(* IEC 61131-3 sources: AXOpen/src/showcase/app/src/IO (part 3) *)

	TYPE
        {S7.extern=ReadWrite}
        {#ix-attr:[Container(Layout.Wrap)]}
	    cognex_insight_7600_ResultData_128_Input_Layout : STRUCT
	        Signals_0 AT %B0 : WORD;
	        Signals_1 AT %B2 : WORD;
	        Signals_2 AT %B4 : ARRAY[0..127] OF BYTE;
	    END_STRUCT;
	END_TYPE

	TYPE
        {S7.extern=ReadWrite}
        {#ix-attr:[Container(Layout.Wrap)]}
	    cognex_insight_7600_SoftEvent_Control_Input_Layout : STRUCT
	        Signals_0 AT %X0.0 : BOOL;
	        Signals_1 AT %X0.1 : BOOL;
	        Signals_2 AT %X0.2 : BOOL;
	        Signals_3 AT %X0.3 : BOOL;
	        Signals_4 AT %X0.4 : BOOL;
	        Signals_5 AT %X0.5 : BOOL;
	        Signals_6 AT %X0.6 : BOOL;
	        Signals_7 AT %X0.7 : BOOL;
	    END_STRUCT;
	END_TYPE

	TYPE
        {S7.extern=ReadWrite}
        {#ix-attr:[Container(Layout.Wrap)]}
	    cognex_insight_7600_SoftEvent_Control_Output_Layout : STRUCT
	        Signals_8 AT %X0.0 : BOOL;
	        Signals_9 AT %X0.1 : BOOL;
	        Signals_10 AT %X0.2 : BOOL;
	        Signals_11 AT %X0.3 : BOOL;
	        Signals_12 AT %X0.4 : BOOL;
	        Signals_13 AT %X0.5 : BOOL;
	        Signals_14 AT %X0.6 : BOOL;
	        Signals_15 AT %X0.7 : BOOL;
	    END_STRUCT;
	END_TYPE

	TYPE
        {S7.extern=ReadWrite}
        {#ix-attr:[Container(Layout.Wrap)]}
	    cognex_insight_7600_UserData_128_Output_Layout : STRUCT
	        Signals_0 AT %B0 : ARRAY[0..127] OF BYTE;
	    END_STRUCT;
	END_TYPE

	TYPE
        {S7.extern=ReadWrite}
        {#ix-attr:[Container(Layout.Wrap)]}
	    desoutter_cvic_ii_Input_1_byte_1_Input_Layout : STRUCT
	        Signals_0 AT %B0 : BYTE;
	    END_STRUCT;
	END_TYPE

	TYPE
        {S7.extern=ReadWrite}
        {#ix-attr:[Container(Layout.Wrap)]}
	    desoutter_cvic_ii_Input_1_byte_2_Input_Layout : STRUCT
	        Signals_0 AT %B0 : BYTE;
	    END_STRUCT;
	END_TYPE

	TYPE
        {S7.extern=ReadWrite}
        {#ix-attr:[Container(Layout.Wrap)]}
	    desoutter_cvic_ii_Input_1_word_1_Input_Layout : STRUCT
	        Signals_0 AT %B0 : WORD;
	    END_STRUCT;
	END_TYPE

	TYPE
        {S7.extern=ReadWrite}
        {#ix-attr:[Container(Layout.Wrap)]}
	    desoutter_cvic_ii_Input_1_word_2_Input_Layout : STRUCT
	        Signals_0 AT %B0 : WORD;
	    END_STRUCT;
	END_TYPE

	TYPE
        {S7.extern=ReadWrite}
        {#ix-attr:[Container(Layout.Wrap)]}
	    desoutter_cvic_ii_Input_2_word_1_Input_Layout : STRUCT
	        Signals_0 AT %B0 : DWORD;
	    END_STRUCT;
	END_TYPE

	TYPE
        {S7.extern=ReadWrite}
        {#ix-attr:[Container(Layout.Wrap)]}
	    desoutter_cvic_ii_Input_2_word_2_Input_Layout : STRUCT
	        Signals_0 AT %B0 : DWORD;
	    END_STRUCT;
	END_TYPE

	TYPE
        {S7.extern=ReadWrite}
        {#ix-attr:[Container(Layout.Wrap)]}
	    desoutter_cvic_ii_Output_1_byte_1_Output_Layout : STRUCT
	        Signals_0 AT %B0 : BYTE;
	    END_STRUCT;
	END_TYPE

	TYPE
        {S7.extern=ReadWrite}
        {#ix-attr:[Container(Layout.Wrap)]}
	    desoutter_cvic_ii_Output_1_byte_2_Output_Layout : STRUCT
	        Signals_0 AT %B0 : BYTE;
	    END_STRUCT;
	END_TYPE

	TYPE
        {S7.extern=ReadWrite}
        {#ix-attr:[Container(Layout.Wrap)]}
	    dukaneiqauto_iQ_to_PLC_Inputs_Input_Layout : STRUCT
	        Signals_0 AT %B0 : DWORD;
	        Signals_1 AT %B4 : DWORD;
	        Signals_2 AT %B8 : DWORD;
	        Signals_3 AT %B12 : DWORD;
	        Signals_4 AT %B16 : DWORD;
	        Signals_5 AT %B20 : DWORD;
	        Signals_6 AT %B24 : DWORD;
	        Signals_7 AT %B28 : DWORD;
	        Signals_8 AT %B32 : DWORD;
	        Signals_9 AT %B36 : DWORD;
	        Signals_10 AT %B40 : DWORD;
	        Signals_11 AT %B44 : DWORD;
	        Signals_12 AT %B48 : DWORD;
	        Signals_13 AT %B52 : DWORD;
	        Signals_14 AT %B56 : DWORD;
	        Signals_15 AT %B60 : DWORD;
	        Signals_16 AT %B64 : DWORD;
	        Signals_17 AT %B68 : DWORD;
	        Signals_18 AT %B72 : DWORD;
	        Signals_19 AT %B76 : DWORD;
	        Signals_20 AT %B80 : DWORD;
	        Signals_21 AT %B84 : DWORD;
	        Signals_22 AT %B88 : DWORD;
	        Signals_23 AT %B92 : DWORD;
	        Signals_24 AT %B96 : DWORD;
	        Signals_25 AT %B100 : DWORD;
	        Signals_26 AT %B104 : DWORD;
	        Signals_27 AT %B108 : DWORD;
	        Signals_28 AT %B112 : DWORD;
	        Signals_29 AT %B116 : DWORD;
	        Signals_30 AT %B120 : DWORD;
	        Signals_31 AT %B124 : DWORD;
	        Signals_32 AT %B128 : DWORD;
	        Signals_33 AT %B132 : DWORD;
	        Signals_34 AT %B136 : DWORD;
	    END_STRUCT;
	END_TYPE

	TYPE
        {S7.extern=ReadWrite}
        {#ix-attr:[Container(Layout.Wrap)]}
	    dukaneiqauto_PLC_to_iQ_Outputs_Output_Layout : STRUCT
	        Signals_0 AT %B0 : DWORD;
	        Signals_1 AT %B4 : DWORD;
	        Signals_2 AT %B8 : DWORD;
	        Signals_3 AT %B12 : DWORD;
	        Signals_4 AT %B16 : DWORD;
	    END_STRUCT;
	END_TYPE

	TYPE
        {S7.extern=ReadWrite}
        {#ix-attr:[Container(Layout.Wrap)]}
	    et200sp_CM_4xIO_Link_RF200_CM_4xIO_Link_V2_2_144I_128O_1_Input_Layout : STRUCT
	        Signals_0 AT %B0 : BYTE;
	        Signals_1 AT %B1 : BYTE;
	        Signals_2 AT %B2 : BYTE;
	        Signals_3 AT %B3 : BYTE;
	        Signals_4 AT %B4 : BYTE;
	        Signals_5 AT %B5 : BYTE;
	        Signals_6 AT %B6 : BYTE;
	        Signals_7 AT %B7 : BYTE;
	        Signals_8 AT %B8 : BYTE;
	        Signals_9 AT %B9 : BYTE;
	        Signals_10 AT %B10 : BYTE;
	        Signals_11 AT %B11 : BYTE;
	        Signals_12 AT %B12 : BYTE;
	        Signals_13 AT %B13 : BYTE;
	        Signals_14 AT %B14 : BYTE;
	        Signals_15 AT %B15 : BYTE;
	        Signals_16 AT %B16 : BYTE;
	        Signals_17 AT %B17 : BYTE;
	        Signals_18 AT %B18 : BYTE;
	        Signals_19 AT %B19 : BYTE;
	        Signals_20 AT %B20 : BYTE;
	        Signals_21 AT %B21 : BYTE;
	        Signals_22 AT %B22 : BYTE;
	        Signals_23 AT %B23 : BYTE;
	        Signals_24 AT %B24 : BYTE;
	        Signals_25 AT %B25 : BYTE;
	        Signals_26 AT %B26 : BYTE;
	        Signals_27 AT %B27 : BYTE;
	        Signals_28 AT %B28 : BYTE;
	        Signals_29 AT %B29 : BYTE;
	        Signals_30 AT %B30 : BYTE;
	        Signals_31 AT %B31 : BYTE;
	        Signals_32 AT %B32 : BYTE;
	        Signals_33 AT %B33 : BYTE;
	        Signals_34 AT %B34 : BYTE;
	        Signals_35 AT %B35 : BYTE;
	        Signals_36 AT %B36 : BYTE;
	        Signals_37 AT %B37 : BYTE;
	        Signals_38 AT %B38 : BYTE;
	        Signals_39 AT %B39 : BYTE;
	        Signals_40 AT %B40 : BYTE;
	        Signals_41 AT %B41 : BYTE;
	        Signals_42 AT %B42 : BYTE;
	        Signals_43 AT %B43 : BYTE;
	        Signals_44 AT %B44 : BYTE;
	        Signals_45 AT %B45 : BYTE;
	        Signals_46 AT %B46 : BYTE;
	        Signals_47 AT %B47 : BYTE;
	        Signals_48 AT %B48 : BYTE;
	        Signals_49 AT %B49 : BYTE;
	        Signals_50 AT %B50 : BYTE;
	        Signals_51 AT %B51 : BYTE;
	        Signals_52 AT %B52 : BYTE;
	        Signals_53 AT %B53 : BYTE;
	        Signals_54 AT %B54 : BYTE;
	        Signals_55 AT %B55 : BYTE;
	        Signals_56 AT %B56 : BYTE;
	        Signals_57 AT %B57 : BYTE;
	        Signals_58 AT %B58 : BYTE;
	        Signals_59 AT %B59 : BYTE;
	        Signals_60 AT %B60 : BYTE;
	        Signals_61 AT %B61 : BYTE;
	        Signals_62 AT %B62 : BYTE;
	        Signals_63 AT %B63 : BYTE;
	        Signals_64 AT %B64 : BYTE;
	        Signals_65 AT %B65 : BYTE;
	        Signals_66 AT %B66 : BYTE;
	        Signals_67 AT %B67 : BYTE;
	        Signals_68 AT %B68 : BYTE;
	        Signals_69 AT %B69 : BYTE;
	        Signals_70 AT %B70 : BYTE;
	        Signals_71 AT %B71 : BYTE;
	        Signals_72 AT %B72 : BYTE;
	        Signals_73 AT %B73 : BYTE;
	        Signals_74 AT %B74 : BYTE;
	        Signals_75 AT %B75 : BYTE;
	        Signals_76 AT %B76 : BYTE;
	        Signals_77 AT %B77 : BYTE;
	        Signals_78 AT %B78 : BYTE;
	        Signals_79 AT %B79 : BYTE;
	        Signals_80 AT %B80 : BYTE;
	        Signals_81 AT %B81 : BYTE;
	        Signals_82 AT %B82 : BYTE;
	        Signals_83 AT %B83 : BYTE;
	        Signals_84 AT %B84 : BYTE;
	        Signals_85 AT %B85 : BYTE;
	        Signals_86 AT %B86 : BYTE;
	        Signals_87 AT %B87 : BYTE;
	        Signals_88 AT %B88 : BYTE;
	        Signals_89 AT %B89 : BYTE;
	        Signals_90 AT %B90 : BYTE;
	        Signals_91 AT %B91 : BYTE;
	        Signals_92 AT %B92 : BYTE;
	        Signals_93 AT %B93 : BYTE;
	        Signals_94 AT %B94 : BYTE;
	        Signals_95 AT %B95 : BYTE;
	        Signals_96 AT %B96 : BYTE;
	        Signals_97 AT %B97 : BYTE;
	        Signals_98 AT %B98 : BYTE;
	        Signals_99 AT %B99 : BYTE;
	        Signals_100 AT %B100 : BYTE;
	        Signals_101 AT %B101 : BYTE;
	        Signals_102 AT %B102 : BYTE;
	        Signals_103 AT %B103 : BYTE;
	        Signals_104 AT %B104 : BYTE;
	        Signals_105 AT %B105 : BYTE;
	        Signals_106 AT %B106 : BYTE;
	        Signals_107 AT %B107 : BYTE;
	        Signals_108 AT %B108 : BYTE;
	        Signals_109 AT %B109 : BYTE;
	        Signals_110 AT %B110 : BYTE;
	        Signals_111 AT %B111 : BYTE;
	        Signals_112 AT %B112 : BYTE;
	        Signals_113 AT %B113 : BYTE;
	        Signals_114 AT %B114 : BYTE;
	        Signals_115 AT %B115 : BYTE;
	        Signals_116 AT %B116 : BYTE;
	        Signals_117 AT %B117 : BYTE;
	        Signals_118 AT %B118 : BYTE;
	        Signals_119 AT %B119 : BYTE;
	        Signals_120 AT %B120 : BYTE;
	        Signals_121 AT %B121 : BYTE;
	        Signals_122 AT %B122 : BYTE;
	        Signals_123 AT %B123 : BYTE;
	        Signals_124 AT %B124 : BYTE;
	        Signals_125 AT %B125 : BYTE;
	        Signals_126 AT %B126 : BYTE;
	        Signals_127 AT %B127 : BYTE;
	        Signals_128 AT %B128 : BYTE;
	        Signals_129 AT %B129 : BYTE;
	        Signals_130 AT %B130 : BYTE;
	        Signals_131 AT %B131 : BYTE;
	        Signals_132 AT %B132 : BYTE;
	        Signals_133 AT %B133 : BYTE;
	        Signals_134 AT %B134 : BYTE;
	        Signals_135 AT %B135 : BYTE;
	        Signals_136 AT %B136 : BYTE;
	        Signals_137 AT %B137 : BYTE;
	        Signals_138 AT %B138 : BYTE;
	        Signals_139 AT %B139 : BYTE;
	        Signals_140 AT %B140 : BYTE;
	        Signals_141 AT %B141 : BYTE;
	        Signals_142 AT %B142 : BYTE;
	        Signals_143 AT %B143 : BYTE;
	    END_STRUCT;
	END_TYPE

	TYPE
        {S7.extern=ReadWrite}
        {#ix-attr:[Container(Layout.Wrap)]}
	    et200sp_CM_4xIO_Link_RF200_CM_4xIO_Link_V2_2_144I_128O_1_Output_Layout : STRUCT
	        Signals_144 AT %B0 : BYTE;
	        Signals_145 AT %B1 : BYTE;
	        Signals_146 AT %B2 : BYTE;
	        Signals_147 AT %B3 : BYTE;
	        Signals_148 AT %B4 : BYTE;
	        Signals_149 AT %B5 : BYTE;
	        Signals_150 AT %B6 : BYTE;
	        Signals_151 AT %B7 : BYTE;
	        Signals_152 AT %B8 : BYTE;
	        Signals_153 AT %B9 : BYTE;
	        Signals_154 AT %B10 : BYTE;
	        Signals_155 AT %B11 : BYTE;
	        Signals_156 AT %B12 : BYTE;
	        Signals_157 AT %B13 : BYTE;
	        Signals_158 AT %B14 : BYTE;
	        Signals_159 AT %B15 : BYTE;
	        Signals_160 AT %B16 : BYTE;
	        Signals_161 AT %B17 : BYTE;
	        Signals_162 AT %B18 : BYTE;
	        Signals_163 AT %B19 : BYTE;
	        Signals_164 AT %B20 : BYTE;
	        Signals_165 AT %B21 : BYTE;
	        Signals_166 AT %B22 : BYTE;
	        Signals_167 AT %B23 : BYTE;
	        Signals_168 AT %B24 : BYTE;
	        Signals_169 AT %B25 : BYTE;
	        Signals_170 AT %B26 : BYTE;
	        Signals_171 AT %B27 : BYTE;
	        Signals_172 AT %B28 : BYTE;
	        Signals_173 AT %B29 : BYTE;
	        Signals_174 AT %B30 : BYTE;
	        Signals_175 AT %B31 : BYTE;
	        Signals_176 AT %B32 : BYTE;
	        Signals_177 AT %B33 : BYTE;
	        Signals_178 AT %B34 : BYTE;
	        Signals_179 AT %B35 : BYTE;
	        Signals_180 AT %B36 : BYTE;
	        Signals_181 AT %B37 : BYTE;
	        Signals_182 AT %B38 : BYTE;
	        Signals_183 AT %B39 : BYTE;
	        Signals_184 AT %B40 : BYTE;
	        Signals_185 AT %B41 : BYTE;
	        Signals_186 AT %B42 : BYTE;
	        Signals_187 AT %B43 : BYTE;
	        Signals_188 AT %B44 : BYTE;
	        Signals_189 AT %B45 : BYTE;
	        Signals_190 AT %B46 : BYTE;
	        Signals_191 AT %B47 : BYTE;
	        Signals_192 AT %B48 : BYTE;
	        Signals_193 AT %B49 : BYTE;
	        Signals_194 AT %B50 : BYTE;
	        Signals_195 AT %B51 : BYTE;
	        Signals_196 AT %B52 : BYTE;
	        Signals_197 AT %B53 : BYTE;
	        Signals_198 AT %B54 : BYTE;
	        Signals_199 AT %B55 : BYTE;
	        Signals_200 AT %B56 : BYTE;
	        Signals_201 AT %B57 : BYTE;
	        Signals_202 AT %B58 : BYTE;
	        Signals_203 AT %B59 : BYTE;
	        Signals_204 AT %B60 : BYTE;
	        Signals_205 AT %B61 : BYTE;
	        Signals_206 AT %B62 : BYTE;
	        Signals_207 AT %B63 : BYTE;
	        Signals_208 AT %B64 : BYTE;
	        Signals_209 AT %B65 : BYTE;
	        Signals_210 AT %B66 : BYTE;
	        Signals_211 AT %B67 : BYTE;
	        Signals_212 AT %B68 : BYTE;
	        Signals_213 AT %B69 : BYTE;
	        Signals_214 AT %B70 : BYTE;
	        Signals_215 AT %B71 : BYTE;
	        Signals_216 AT %B72 : BYTE;
	        Signals_217 AT %B73 : BYTE;
	        Signals_218 AT %B74 : BYTE;
	        Signals_219 AT %B75 : BYTE;
	        Signals_220 AT %B76 : BYTE;
	        Signals_221 AT %B77 : BYTE;
	        Signals_222 AT %B78 : BYTE;
	        Signals_223 AT %B79 : BYTE;
	        Signals_224 AT %B80 : BYTE;
	        Signals_225 AT %B81 : BYTE;
	        Signals_226 AT %B82 : BYTE;
	        Signals_227 AT %B83 : BYTE;
	        Signals_228 AT %B84 : BYTE;
	        Signals_229 AT %B85 : BYTE;
	        Signals_230 AT %B86 : BYTE;
	        Signals_231 AT %B87 : BYTE;
	        Signals_232 AT %B88 : BYTE;
	        Signals_233 AT %B89 : BYTE;
	        Signals_234 AT %B90 : BYTE;
	        Signals_235 AT %B91 : BYTE;
	        Signals_236 AT %B92 : BYTE;
	        Signals_237 AT %B93 : BYTE;
	        Signals_238 AT %B94 : BYTE;
	        Signals_239 AT %B95 : BYTE;
	        Signals_240 AT %B96 : BYTE;
	        Signals_241 AT %B97 : BYTE;
	        Signals_242 AT %B98 : BYTE;
	        Signals_243 AT %B99 : BYTE;
	        Signals_244 AT %B100 : BYTE;
	        Signals_245 AT %B101 : BYTE;
	        Signals_246 AT %B102 : BYTE;
	        Signals_247 AT %B103 : BYTE;
	        Signals_248 AT %B104 : BYTE;
	        Signals_249 AT %B105 : BYTE;
	        Signals_250 AT %B106 : BYTE;
	        Signals_251 AT %B107 : BYTE;
	        Signals_252 AT %B108 : BYTE;
	        Signals_253 AT %B109 : BYTE;
	        Signals_254 AT %B110 : BYTE;
	        Signals_255 AT %B111 : BYTE;
	        Signals_256 AT %B112 : BYTE;
	        Signals_257 AT %B113 : BYTE;
	        Signals_258 AT %B114 : BYTE;
	        Signals_259 AT %B115 : BYTE;
	        Signals_260 AT %B116 : BYTE;
	        Signals_261 AT %B117 : BYTE;
	        Signals_262 AT %B118 : BYTE;
	        Signals_263 AT %B119 : BYTE;
	        Signals_264 AT %B120 : BYTE;
	        Signals_265 AT %B121 : BYTE;
	        Signals_266 AT %B122 : BYTE;
	        Signals_267 AT %B123 : BYTE;
	        Signals_268 AT %B124 : BYTE;
	        Signals_269 AT %B125 : BYTE;
	        Signals_270 AT %B126 : BYTE;
	        Signals_271 AT %B127 : BYTE;
	    END_STRUCT;
	END_TYPE

	TYPE
        {S7.extern=ReadWrite}
        {#ix-attr:[Container(Layout.Wrap)]}
	    et200sp_CpPtp_Input_Layout : STRUCT
	        Signals_0 AT %B0 : BYTE;
	        Signals_1 AT %B1 : BYTE;
	        Signals_2 AT %B2 : BYTE;
	        Signals_3 AT %B3 : BYTE;
	        Signals_4 AT %B4 : BYTE;
	        Signals_5 AT %B5 : BYTE;
	        Signals_6 AT %B6 : BYTE;
	        Signals_7 AT %B7 : BYTE;
	    END_STRUCT;
	END_TYPE

	TYPE
        {S7.extern=ReadWrite}
        {#ix-attr:[Container(Layout.Wrap)]}
	    festo_cmmtas_DoServo_SiemensTelegram111_PZD_12_12_Input_Layout : STRUCT
	        Signals_0 AT %X0.0 : BOOL;
	        Signals_1 AT %X0.1 : BOOL;
	        Signals_2 AT %X0.2 : BOOL;
	        Signals_3 AT %X0.3 : BOOL;
	        Signals_4 AT %X0.4 : BOOL;
	        Signals_5 AT %X0.5 : BOOL;
	        Signals_6 AT %X0.6 : BOOL;
	        Signals_7 AT %X0.7 : BOOL;
	        Signals_8 AT %X1.0 : BOOL;
	        Signals_9 AT %X1.1 : BOOL;
	        Signals_10 AT %X1.2 : BOOL;
	        Signals_11 AT %X1.3 : BOOL;
	        Signals_12 AT %X1.4 : BOOL;
	        Signals_13 AT %X1.5 : BOOL;
	        Signals_14 AT %X1.6 : BOOL;
	        Signals_15 AT %X1.7 : BOOL;
	        Signals_16 AT %X2.0 : BOOL;
	        Signals_17 AT %X2.1 : BOOL;
	        Signals_18 AT %X2.2 : BOOL;
	        Signals_19 AT %X2.3 : BOOL;
	        Signals_20 AT %X2.4 : BOOL;
	        Signals_21 AT %X2.5 : BOOL;
	        Signals_22 AT %X2.6 : BOOL;
	        Signals_23 AT %X2.7 : BOOL;
	        Signals_24 AT %X3.0 : BOOL;
	        Signals_25 AT %X3.1 : BOOL;
	        Signals_26 AT %X3.2 : BOOL;
	        Signals_27 AT %X3.3 : BOOL;
	        Signals_28 AT %X3.4 : BOOL;
	        Signals_29 AT %X3.5 : BOOL;
	        Signals_30 AT %X3.6 : BOOL;
	        Signals_31 AT %X3.7 : BOOL;
	        Signals_32 AT %X4.0 : BOOL;
	        Signals_33 AT %X4.1 : BOOL;
	        Signals_34 AT %X4.2 : BOOL;
	        Signals_35 AT %X4.3 : BOOL;
	        Signals_36 AT %X4.4 : BOOL;
	        Signals_37 AT %X4.5 : BOOL;
	        Signals_38 AT %X4.6 : BOOL;
	        Signals_39 AT %X4.7 : BOOL;
	        Signals_40 AT %X5.0 : BOOL;
	        Signals_41 AT %X5.1 : BOOL;
	        Signals_42 AT %X5.2 : BOOL;
	        Signals_43 AT %X5.3 : BOOL;
	        Signals_44 AT %X5.4 : BOOL;
	        Signals_45 AT %X5.5 : BOOL;
	        Signals_46 AT %X5.6 : BOOL;
	        Signals_47 AT %X5.7 : BOOL;
	        Signals_48 AT %X6.0 : BOOL;
	        Signals_49 AT %X6.1 : BOOL;
	        Signals_50 AT %X6.2 : BOOL;
	        Signals_51 AT %X6.3 : BOOL;
	        Signals_52 AT %X6.4 : BOOL;
	        Signals_53 AT %X6.5 : BOOL;
	        Signals_54 AT %X6.6 : BOOL;
	        Signals_55 AT %X6.7 : BOOL;
	        Signals_56 AT %X7.0 : BOOL;
	        Signals_57 AT %X7.1 : BOOL;
	        Signals_58 AT %X7.2 : BOOL;
	        Signals_59 AT %X7.3 : BOOL;
	        Signals_60 AT %X7.4 : BOOL;
	        Signals_61 AT %X7.5 : BOOL;
	        Signals_62 AT %X7.6 : BOOL;
	        Signals_63 AT %X7.7 : BOOL;
	        Signals_64 AT %X8.0 : BOOL;
	        Signals_65 AT %X8.1 : BOOL;
	        Signals_66 AT %X8.2 : BOOL;
	        Signals_67 AT %X8.3 : BOOL;
	        Signals_68 AT %X8.4 : BOOL;
	        Signals_69 AT %X8.5 : BOOL;
	        Signals_70 AT %X8.6 : BOOL;
	        Signals_71 AT %X8.7 : BOOL;
	        Signals_72 AT %X9.0 : BOOL;
	        Signals_73 AT %X9.1 : BOOL;
	        Signals_74 AT %X9.2 : BOOL;
	        Signals_75 AT %X9.3 : BOOL;
	        Signals_76 AT %X9.4 : BOOL;
	        Signals_77 AT %X9.5 : BOOL;
	        Signals_78 AT %X9.6 : BOOL;
	        Signals_79 AT %X9.7 : BOOL;
	        Signals_80 AT %B10 : DWORD;
	        Signals_81 AT %B14 : DWORD;
	        Signals_82 AT %B18 : WORD;
	        Signals_83 AT %B20 : WORD;
	        Signals_84 AT %B22 : WORD;
	    END_STRUCT;
	END_TYPE

	TYPE
        {S7.extern=ReadWrite}
        {#ix-attr:[Container(Layout.Wrap)]}
	    festo_cmmtas_DoServo_SiemensTelegram111_PZD_12_12_Output_Layout : STRUCT
	        Signals_85 AT %X0.0 : BOOL;
	        Signals_86 AT %X0.1 : BOOL;
	        Signals_87 AT %X0.2 : BOOL;
	        Signals_88 AT %X0.3 : BOOL;
	        Signals_89 AT %X0.4 : BOOL;
	        Signals_90 AT %X0.5 : BOOL;
	        Signals_91 AT %X0.6 : BOOL;
	        Signals_92 AT %X0.7 : BOOL;
	        Signals_93 AT %X1.0 : BOOL;
	        Signals_94 AT %X1.1 : BOOL;
	        Signals_95 AT %X1.2 : BOOL;
	        Signals_96 AT %X1.3 : BOOL;
	        Signals_97 AT %X1.4 : BOOL;
	        Signals_98 AT %X1.5 : BOOL;
	        Signals_99 AT %X1.6 : BOOL;
	        Signals_100 AT %X1.7 : BOOL;
	        Signals_101 AT %X2.0 : BOOL;
	        Signals_102 AT %X2.1 : BOOL;
	        Signals_103 AT %X2.2 : BOOL;
	        Signals_104 AT %X2.3 : BOOL;
	        Signals_105 AT %X2.4 : BOOL;
	        Signals_106 AT %X2.5 : BOOL;
	        Signals_107 AT %X2.6 : BOOL;
	        Signals_108 AT %X2.7 : BOOL;
	        Signals_109 AT %X3.0 : BOOL;
	        Signals_110 AT %X3.1 : BOOL;
	        Signals_111 AT %X3.2 : BOOL;
	        Signals_112 AT %X3.3 : BOOL;
	        Signals_113 AT %X3.4 : BOOL;
	        Signals_114 AT %X3.5 : BOOL;
	        Signals_115 AT %X3.6 : BOOL;
	        Signals_116 AT %X3.7 : BOOL;
	        Signals_117 AT %X4.0 : BOOL;
	        Signals_118 AT %X4.1 : BOOL;
	        Signals_119 AT %X4.2 : BOOL;
	        Signals_120 AT %X4.3 : BOOL;
	        Signals_121 AT %X4.4 : BOOL;
	        Signals_122 AT %X4.5 : BOOL;
	        Signals_123 AT %X4.6 : BOOL;
	        Signals_124 AT %X4.7 : BOOL;
	        Signals_125 AT %X5.0 : BOOL;
	        Signals_126 AT %X5.1 : BOOL;
	        Signals_127 AT %X5.2 : BOOL;
	        Signals_128 AT %X5.3 : BOOL;
	        Signals_129 AT %X5.4 : BOOL;
	        Signals_130 AT %X5.5 : BOOL;
	        Signals_131 AT %X5.6 : BOOL;
	        Signals_132 AT %X5.7 : BOOL;
	        Signals_133 AT %X6.0 : BOOL;
	        Signals_134 AT %X6.1 : BOOL;
	        Signals_135 AT %X6.2 : BOOL;
	        Signals_136 AT %X6.3 : BOOL;
	        Signals_137 AT %X6.4 : BOOL;
	        Signals_138 AT %X6.5 : BOOL;
	        Signals_139 AT %X6.6 : BOOL;
	        Signals_140 AT %X6.7 : BOOL;
	        Signals_141 AT %X7.0 : BOOL;
	        Signals_142 AT %X7.1 : BOOL;
	        Signals_143 AT %X7.2 : BOOL;
	        Signals_144 AT %X7.3 : BOOL;
	        Signals_145 AT %X7.4 : BOOL;
	        Signals_146 AT %X7.5 : BOOL;
	        Signals_147 AT %X7.6 : BOOL;
	        Signals_148 AT %X7.7 : BOOL;
	        Signals_149 AT %B8 : WORD;
	        Signals_150 AT %B10 : DINT;
	        Signals_151 AT %B14 : DWORD;
	        Signals_152 AT %B18 : WORD;
	        Signals_153 AT %B20 : WORD;
	        Signals_154 AT %B22 : WORD;
	    END_STRUCT;
	END_TYPE

	TYPE
        {S7.extern=ReadWrite}
        {#ix-attr:[Container(Layout.Wrap)]}
	    festo_cmmtas_DoServo_SiemensTelegram750_PZD_4_1_Input_Layout : STRUCT
	        Signals_0 AT %B0 : WORD;
	    END_STRUCT;
	END_TYPE

	TYPE
        {S7.extern=ReadWrite}
        {#ix-attr:[Container(Layout.Wrap)]}
	    festo_cmmtas_DoServo_SiemensTelegram750_PZD_4_1_Output_Layout : STRUCT
	        Signals_1 AT %B0 : WORD;
	        Signals_2 AT %B2 : WORD;
	        Signals_3 AT %B4 : WORD;
	        Signals_4 AT %B6 : WORD;
	    END_STRUCT;
	END_TYPE

	TYPE
        {S7.extern=ReadWrite}
        {#ix-attr:[Container(Layout.Wrap)]}
	    keyence_iv3_CommandControl_Output_Layout : STRUCT
	        Signals_0 AT %X0.0 : BOOL;
	        Signals_1 AT %X0.1 : BOOL;
	        Signals_2 AT %X0.2 : BOOL;
	        Signals_3 AT %X0.3 : BOOL;
	        Signals_4 AT %X0.4 : BOOL;
	        Signals_5 AT %X0.5 : BOOL;
	        Signals_6 AT %X0.6 : BOOL;
	        Signals_7 AT %X0.7 : BOOL;
	        Signals_8 AT %B1 : BYTE;
	        Signals_9 AT %X2.0 : BOOL;
	        Signals_10 AT %B3 : BYTE;
	        Signals_11 AT %B4 : WORD;
	        Signals_12 AT %B6 : WORD;
	        Signals_13 AT %B8 : DWORD;
	    END_STRUCT;
	END_TYPE

	TYPE
        {S7.extern=ReadWrite}
        {#ix-attr:[Container(Layout.Wrap)]}
	    keyence_iv3_CommandStatusBits_Input_Layout : STRUCT
	        Signals_0 AT %X0.0 : BOOL;
	        Signals_1 AT %X0.1 : BOOL;
	        Signals_2 AT %X0.2 : BOOL;
	        Signals_3 AT %X0.3 : BOOL;
	        Signals_4 AT %X0.4 : BOOL;
	        Signals_5 AT %X0.5 : BOOL;
	        Signals_6 AT %X0.6 : BOOL;
	        Signals_7 AT %X0.7 : BOOL;
	        Signals_8 AT %X1.0 : BOOL;
	        Signals_9 AT %X1.1 : BOOL;
	        Signals_10 AT %X1.2 : BOOL;
	        Signals_11 AT %X1.6 : BOOL;
	        Signals_12 AT %X1.7 : BOOL;
	        Signals_13 AT %X2.0 : BOOL;
	        Signals_14 AT %X2.1 : BOOL;
	        Signals_15 AT %X2.2 : BOOL;
	        Signals_16 AT %X2.3 : BOOL;
	        Signals_17 AT %X2.4 : BOOL;
	        Signals_18 AT %X2.5 : BOOL;
	        Signals_19 AT %X2.7 : BOOL;
	        Signals_20 AT %X3.0 : BOOL;
	        Signals_21 AT %X3.4 : BOOL;
	        Signals_22 AT %X3.5 : BOOL;
	        Signals_23 AT %X3.6 : BOOL;
	        Signals_24 AT %X3.7 : BOOL;
	    END_STRUCT;
	END_TYPE

	TYPE
        {S7.extern=ReadWrite}
        {#ix-attr:[Container(Layout.Wrap)]}
	    keyence_iv3_DeviceResultBits_1_Input_Layout : STRUCT
	        Signals_0 AT %X0.0 : BOOL;
	        Signals_1 AT %X0.1 : BOOL;
	        Signals_2 AT %X0.2 : BOOL;
	        Signals_3 AT %X0.3 : BOOL;
	        Signals_4 AT %X0.4 : BOOL;
	        Signals_5 AT %X0.5 : BOOL;
	        Signals_6 AT %X0.6 : BOOL;
	        Signals_7 AT %B1 : BYTE;
	        Signals_8 AT %X2.0 : BOOL;
	        Signals_9 AT %X2.1 : BOOL;
	        Signals_10 AT %X2.2 : BOOL;
	        Signals_11 AT %X2.3 : BOOL;
	        Signals_12 AT %X2.4 : BOOL;
	        Signals_13 AT %X2.5 : BOOL;
	        Signals_14 AT %X2.6 : BOOL;
	        Signals_15 AT %X2.7 : BOOL;
	        Signals_16 AT %X3.0 : BOOL;
	        Signals_17 AT %X3.1 : BOOL;
	        Signals_18 AT %X3.2 : BOOL;
	        Signals_19 AT %X3.3 : BOOL;
	        Signals_20 AT %X3.4 : BOOL;
	        Signals_21 AT %X3.5 : BOOL;
	        Signals_22 AT %X3.6 : BOOL;
	        Signals_23 AT %X3.7 : BOOL;
	    END_STRUCT;
	END_TYPE

	TYPE
        {S7.extern=ReadWrite}
        {#ix-attr:[Container(Layout.Wrap)]}
	    keyence_iv3_DeviceResultBits_2_Input_Layout : STRUCT
	        Signals_0 AT %B0 : WORD;
	        Signals_1 AT %X2.0 : BOOL;
	        Signals_2 AT %X2.1 : BOOL;
	        Signals_3 AT %X2.2 : BOOL;
	        Signals_4 AT %X2.3 : BOOL;
	        Signals_5 AT %X2.4 : BOOL;
	        Signals_6 AT %X2.5 : BOOL;
	        Signals_7 AT %X2.6 : BOOL;
	        Signals_8 AT %X2.7 : BOOL;
	        Signals_9 AT %X3.0 : BOOL;
	        Signals_10 AT %X3.1 : BOOL;
	        Signals_11 AT %X3.2 : BOOL;
	        Signals_12 AT %X3.3 : BOOL;
	        Signals_13 AT %X3.4 : BOOL;
	        Signals_14 AT %X3.5 : BOOL;
	        Signals_15 AT %X3.6 : BOOL;
	        Signals_16 AT %X3.7 : BOOL;
	        Signals_17 AT %X4.0 : BOOL;
	        Signals_18 AT %X4.1 : BOOL;
	        Signals_19 AT %X4.2 : BOOL;
	        Signals_20 AT %X4.3 : BOOL;
	        Signals_21 AT %X4.4 : BOOL;
	        Signals_22 AT %X4.5 : BOOL;
	        Signals_23 AT %X4.6 : BOOL;
	        Signals_24 AT %X4.7 : BOOL;
	        Signals_25 AT %X5.0 : BOOL;
	        Signals_26 AT %X5.1 : BOOL;
	        Signals_27 AT %X5.2 : BOOL;
	        Signals_28 AT %X5.3 : BOOL;
	        Signals_29 AT %X5.4 : BOOL;
	        Signals_30 AT %X5.5 : BOOL;
	        Signals_31 AT %X5.6 : BOOL;
	        Signals_32 AT %X5.7 : BOOL;
	        Signals_33 AT %X6.0 : BOOL;
	        Signals_34 AT %X6.1 : BOOL;
	        Signals_35 AT %X6.2 : BOOL;
	        Signals_36 AT %X6.3 : BOOL;
	        Signals_37 AT %X6.4 : BOOL;
	        Signals_38 AT %X6.5 : BOOL;
	        Signals_39 AT %X6.6 : BOOL;
	        Signals_40 AT %X6.7 : BOOL;
	        Signals_41 AT %X7.0 : BOOL;
	        Signals_42 AT %X7.1 : BOOL;
	        Signals_43 AT %X7.2 : BOOL;
	        Signals_44 AT %X7.3 : BOOL;
	        Signals_45 AT %X7.4 : BOOL;
	        Signals_46 AT %X7.5 : BOOL;
	        Signals_47 AT %X7.6 : BOOL;
	        Signals_48 AT %X7.7 : BOOL;
	    END_STRUCT;
	END_TYPE

	TYPE
        {S7.extern=ReadWrite}
        {#ix-attr:[Container(Layout.Wrap)]}
	    keyence_iv3_DeviceStatistics_Input_Layout : STRUCT
	        Signals_0 AT %B0 : WORD;
	        Signals_1 AT %B2 : WORD;
	        Signals_2 AT %B4 : WORD;
	        Signals_3 AT %B6 : WORD;
	        Signals_4 AT %B8 : DWORD;
	        Signals_5 AT %B12 : DWORD;
	        Signals_6 AT %B16 : DWORD;
	        Signals_7 AT %B20 : DWORD;
	        Signals_8 AT %B24 : DWORD;
	    END_STRUCT;
	END_TYPE

	TYPE
        {S7.extern=ReadWrite}
        {#ix-attr:[Container(Layout.Wrap)]}
	    keyence_iv3_DeviceStatusWords_Input_Layout : STRUCT
	        Signals_0 AT %B0 : WORD;
	        Signals_1 AT %B2 : WORD;
	        Signals_2 AT %B4 : WORD;
	        Signals_3 AT %B6 : WORD;
	        Signals_4 AT %B8 : WORD;
	        Signals_5 AT %B10 : WORD;
	        Signals_6 AT %B12 : WORD;
	        Signals_7 AT %B14 : WORD;
	    END_STRUCT;
	END_TYPE

	TYPE
        {S7.extern=ReadWrite}
        {#ix-attr:[Container(Layout.Wrap)]}
	    keyence_iv3_PositionAdjustResult_Input_Layout : STRUCT
	        Signals_0 AT %B0 : WORD;
	        Signals_1 AT %B2 : WORD;
	        Signals_2 AT %B4 : WORD;
	        Signals_3 AT %B6 : WORD;
	        Signals_4 AT %B8 : WORD;
	        Signals_5 AT %B10 : WORD;
	        Signals_6 AT %B12 : WORD;
	        Signals_7 AT %B14 : WORD;
	        Signals_8 AT %B16 : WORD;
	        Signals_9 AT %B18 : WORD;
	    END_STRUCT;
	END_TYPE

	TYPE
        {S7.extern=ReadWrite}
        {#ix-attr:[Container(Layout.Wrap)]}
	    keyence_iv3_ToolResult_1_Input_Layout : STRUCT
	        Signals_0 AT %B0 : WORD;
	        Signals_1 AT %B2 : WORD;
	        Signals_2 AT %B4 : WORD;
	        Signals_3 AT %B6 : WORD;
	        Signals_4 AT %B8 : WORD;
	        Signals_5 AT %B10 : WORD;
	        Signals_6 AT %B12 : WORD;
	        Signals_7 AT %B14 : WORD;
	        Signals_8 AT %B16 : WORD;
	        Signals_9 AT %B18 : WORD;
	    END_STRUCT;
	END_TYPE

	TYPE
        {S7.extern=ReadWrite}
        {#ix-attr:[Container(Layout.Wrap)]}
	    keyence_iv3_ToolResult_10_Input_Layout : STRUCT
	        Signals_0 AT %B0 : WORD;
	        Signals_1 AT %B2 : WORD;
	        Signals_2 AT %B4 : WORD;
	        Signals_3 AT %B6 : WORD;
	        Signals_4 AT %B8 : WORD;
	        Signals_5 AT %B10 : WORD;
	        Signals_6 AT %B12 : WORD;
	        Signals_7 AT %B14 : WORD;
	        Signals_8 AT %B16 : WORD;
	        Signals_9 AT %B18 : WORD;
	    END_STRUCT;
	END_TYPE

	TYPE
        {S7.extern=ReadWrite}
        {#ix-attr:[Container(Layout.Wrap)]}
	    keyence_iv3_ToolResult_11_Input_Layout : STRUCT
	        Signals_0 AT %B0 : WORD;
	        Signals_1 AT %B2 : WORD;
	        Signals_2 AT %B4 : WORD;
	        Signals_3 AT %B6 : WORD;
	        Signals_4 AT %B8 : WORD;
	        Signals_5 AT %B10 : WORD;
	        Signals_6 AT %B12 : WORD;
	        Signals_7 AT %B14 : WORD;
	        Signals_8 AT %B16 : WORD;
	        Signals_9 AT %B18 : WORD;
	    END_STRUCT;
	END_TYPE

	TYPE
        {S7.extern=ReadWrite}
        {#ix-attr:[Container(Layout.Wrap)]}
	    keyence_iv3_ToolResult_12_Input_Layout : STRUCT
	        Signals_0 AT %B0 : WORD;
	        Signals_1 AT %B2 : WORD;
	        Signals_2 AT %B4 : WORD;
	        Signals_3 AT %B6 : WORD;
	        Signals_4 AT %B8 : WORD;
	        Signals_5 AT %B10 : WORD;
	        Signals_6 AT %B12 : WORD;
	        Signals_7 AT %B14 : WORD;
	        Signals_8 AT %B16 : WORD;
	        Signals_9 AT %B18 : WORD;
	    END_STRUCT;
	END_TYPE

	TYPE
        {S7.extern=ReadWrite}
        {#ix-attr:[Container(Layout.Wrap)]}
	    keyence_iv3_ToolResult_13_Input_Layout : STRUCT
	        Signals_0 AT %B0 : WORD;
	        Signals_1 AT %B2 : WORD;
	        Signals_2 AT %B4 : WORD;
	        Signals_3 AT %B6 : WORD;
	        Signals_4 AT %B8 : WORD;
	        Signals_5 AT %B10 : WORD;
	        Signals_6 AT %B12 : WORD;
	        Signals_7 AT %B14 : WORD;
	        Signals_8 AT %B16 : WORD;
	        Signals_9 AT %B18 : WORD;
	    END_STRUCT;
	END_TYPE

	TYPE
        {S7.extern=ReadWrite}
        {#ix-attr:[Container(Layout.Wrap)]}
	    keyence_iv3_ToolResult_14_Input_Layout : STRUCT
	        Signals_0 AT %B0 : WORD;
	        Signals_1 AT %B2 : WORD;
	        Signals_2 AT %B4 : WORD;
	        Signals_3 AT %B6 : WORD;
	        Signals_4 AT %B8 : WORD;
	        Signals_5 AT %B10 : WORD;
	        Signals_6 AT %B12 : WORD;
	        Signals_7 AT %B14 : WORD;
	        Signals_8 AT %B16 : WORD;
	        Signals_9 AT %B18 : WORD;
	    END_STRUCT;
	END_TYPE

	TYPE
        {S7.extern=ReadWrite}
        {#ix-attr:[Container(Layout.Wrap)]}
	    keyence_iv3_ToolResult_15_Input_Layout : STRUCT
	        Signals_0 AT %B0 : WORD;
	        Signals_1 AT %B2 : WORD;
	        Signals_2 AT %B4 : WORD;
	        Signals_3 AT %B6 : WORD;
	        Signals_4 AT %B8 : WORD;
	        Signals_5 AT %B10 : WORD;
	        Signals_6 AT %B12 : WORD;
	        Signals_7 AT %B14 : WORD;
	        Signals_8 AT %B16 : WORD;
	        Signals_9 AT %B18 : WORD;
	    END_STRUCT;
	END_TYPE

	TYPE
        {S7.extern=ReadWrite}
        {#ix-attr:[Container(Layout.Wrap)]}
	    keyence_iv3_ToolResult_16_Input_Layout : STRUCT
	        Signals_0 AT %B0 : WORD;
	        Signals_1 AT %B2 : WORD;
	        Signals_2 AT %B4 : WORD;
	        Signals_3 AT %B6 : WORD;
	        Signals_4 AT %B8 : WORD;
	        Signals_5 AT %B10 : WORD;
	        Signals_6 AT %B12 : WORD;
	        Signals_7 AT %B14 : WORD;
	        Signals_8 AT %B16 : WORD;
	        Signals_9 AT %B18 : WORD;
	    END_STRUCT;
	END_TYPE

	TYPE
        {S7.extern=ReadWrite}
        {#ix-attr:[Container(Layout.Wrap)]}
	    keyence_iv3_ToolResult_17_Input_Layout : STRUCT
	        Signals_0 AT %B0 : WORD;
	        Signals_1 AT %B2 : WORD;
	        Signals_2 AT %B4 : WORD;
	        Signals_3 AT %B6 : WORD;
	        Signals_4 AT %B8 : WORD;
	        Signals_5 AT %B10 : WORD;
	        Signals_6 AT %B12 : WORD;
	        Signals_7 AT %B14 : WORD;
	        Signals_8 AT %B16 : WORD;
	        Signals_9 AT %B18 : WORD;
	    END_STRUCT;
	END_TYPE

	TYPE
        {S7.extern=ReadWrite}
        {#ix-attr:[Container(Layout.Wrap)]}
	    keyence_iv3_ToolResult_18_Input_Layout : STRUCT
	        Signals_0 AT %B0 : WORD;
	        Signals_1 AT %B2 : WORD;
	        Signals_2 AT %B4 : WORD;
	        Signals_3 AT %B6 : WORD;
	        Signals_4 AT %B8 : WORD;
	        Signals_5 AT %B10 : WORD;
	        Signals_6 AT %B12 : WORD;
	        Signals_7 AT %B14 : WORD;
	        Signals_8 AT %B16 : WORD;
	        Signals_9 AT %B18 : WORD;
	    END_STRUCT;
	END_TYPE

	TYPE
        {S7.extern=ReadWrite}
        {#ix-attr:[Container(Layout.Wrap)]}
	    keyence_iv3_ToolResult_19_Input_Layout : STRUCT
	        Signals_0 AT %B0 : WORD;
	        Signals_1 AT %B2 : WORD;
	        Signals_2 AT %B4 : WORD;
	        Signals_3 AT %B6 : WORD;
	        Signals_4 AT %B8 : WORD;
	        Signals_5 AT %B10 : WORD;
	        Signals_6 AT %B12 : WORD;
	        Signals_7 AT %B14 : WORD;
	        Signals_8 AT %B16 : WORD;
	        Signals_9 AT %B18 : WORD;
	    END_STRUCT;
	END_TYPE

	TYPE
        {S7.extern=ReadWrite}
        {#ix-attr:[Container(Layout.Wrap)]}
	    keyence_iv3_ToolResult_2_Input_Layout : STRUCT
	        Signals_0 AT %B0 : WORD;
	        Signals_1 AT %B2 : WORD;
	        Signals_2 AT %B4 : WORD;
	        Signals_3 AT %B6 : WORD;
	        Signals_4 AT %B8 : WORD;
	        Signals_5 AT %B10 : WORD;
	        Signals_6 AT %B12 : WORD;
	        Signals_7 AT %B14 : WORD;
	        Signals_8 AT %B16 : WORD;
	        Signals_9 AT %B18 : WORD;
	    END_STRUCT;
	END_TYPE

	TYPE
        {S7.extern=ReadWrite}
        {#ix-attr:[Container(Layout.Wrap)]}
	    keyence_iv3_ToolResult_20_Input_Layout : STRUCT
	        Signals_0 AT %B0 : WORD;
	        Signals_1 AT %B2 : WORD;
	        Signals_2 AT %B4 : WORD;
	        Signals_3 AT %B6 : WORD;
	        Signals_4 AT %B8 : WORD;
	        Signals_5 AT %B10 : WORD;
	        Signals_6 AT %B12 : WORD;
	        Signals_7 AT %B14 : WORD;
	        Signals_8 AT %B16 : WORD;
	        Signals_9 AT %B18 : WORD;
	    END_STRUCT;
	END_TYPE

	TYPE
        {S7.extern=ReadWrite}
        {#ix-attr:[Container(Layout.Wrap)]}
	    keyence_iv3_ToolResult_21_Input_Layout : STRUCT
	        Signals_0 AT %B0 : WORD;
	        Signals_1 AT %B2 : WORD;
	        Signals_2 AT %B4 : WORD;
	        Signals_3 AT %B6 : WORD;
	        Signals_4 AT %B8 : WORD;
	        Signals_5 AT %B10 : WORD;
	        Signals_6 AT %B12 : WORD;
	        Signals_7 AT %B14 : WORD;
	        Signals_8 AT %B16 : WORD;
	        Signals_9 AT %B18 : WORD;
	    END_STRUCT;
	END_TYPE

	TYPE
        {S7.extern=ReadWrite}
        {#ix-attr:[Container(Layout.Wrap)]}
	    keyence_iv3_ToolResult_22_Input_Layout : STRUCT
	        Signals_0 AT %B0 : WORD;
	        Signals_1 AT %B2 : WORD;
	        Signals_2 AT %B4 : WORD;
	        Signals_3 AT %B6 : WORD;
	        Signals_4 AT %B8 : WORD;
	        Signals_5 AT %B10 : WORD;
	        Signals_6 AT %B12 : WORD;
	        Signals_7 AT %B14 : WORD;
	        Signals_8 AT %B16 : WORD;
	        Signals_9 AT %B18 : WORD;
	    END_STRUCT;
	END_TYPE

	TYPE
        {S7.extern=ReadWrite}
        {#ix-attr:[Container(Layout.Wrap)]}
	    keyence_iv3_ToolResult_23_Input_Layout : STRUCT
	        Signals_0 AT %B0 : WORD;
	        Signals_1 AT %B2 : WORD;
	        Signals_2 AT %B4 : WORD;
	        Signals_3 AT %B6 : WORD;
	        Signals_4 AT %B8 : WORD;
	        Signals_5 AT %B10 : WORD;
	        Signals_6 AT %B12 : WORD;
	        Signals_7 AT %B14 : WORD;
	        Signals_8 AT %B16 : WORD;
	        Signals_9 AT %B18 : WORD;
	    END_STRUCT;
	END_TYPE

	TYPE
        {S7.extern=ReadWrite}
        {#ix-attr:[Container(Layout.Wrap)]}
	    keyence_iv3_ToolResult_24_Input_Layout : STRUCT
	        Signals_0 AT %B0 : WORD;
	        Signals_1 AT %B2 : WORD;
	        Signals_2 AT %B4 : WORD;
	        Signals_3 AT %B6 : WORD;
	        Signals_4 AT %B8 : WORD;
	        Signals_5 AT %B10 : WORD;
	        Signals_6 AT %B12 : WORD;
	        Signals_7 AT %B14 : WORD;
	        Signals_8 AT %B16 : WORD;
	        Signals_9 AT %B18 : WORD;
	    END_STRUCT;
	END_TYPE

	TYPE
        {S7.extern=ReadWrite}
        {#ix-attr:[Container(Layout.Wrap)]}
	    keyence_iv3_ToolResult_25_Input_Layout : STRUCT
	        Signals_0 AT %B0 : WORD;
	        Signals_1 AT %B2 : WORD;
	        Signals_2 AT %B4 : WORD;
	        Signals_3 AT %B6 : WORD;
	        Signals_4 AT %B8 : WORD;
	        Signals_5 AT %B10 : WORD;
	        Signals_6 AT %B12 : WORD;
	        Signals_7 AT %B14 : WORD;
	        Signals_8 AT %B16 : WORD;
	        Signals_9 AT %B18 : WORD;
	    END_STRUCT;
	END_TYPE

	TYPE
        {S7.extern=ReadWrite}
        {#ix-attr:[Container(Layout.Wrap)]}
	    keyence_iv3_ToolResult_26_Input_Layout : STRUCT
	        Signals_0 AT %B0 : WORD;
	        Signals_1 AT %B2 : WORD;
	        Signals_2 AT %B4 : WORD;
	        Signals_3 AT %B6 : WORD;
	        Signals_4 AT %B8 : WORD;
	        Signals_5 AT %B10 : WORD;
	        Signals_6 AT %B12 : WORD;
	        Signals_7 AT %B14 : WORD;
	        Signals_8 AT %B16 : WORD;
	        Signals_9 AT %B18 : WORD;
	    END_STRUCT;
	END_TYPE

	TYPE
        {S7.extern=ReadWrite}
        {#ix-attr:[Container(Layout.Wrap)]}
	    keyence_iv3_ToolResult_27_Input_Layout : STRUCT
	        Signals_0 AT %B0 : WORD;
	        Signals_1 AT %B2 : WORD;
	        Signals_2 AT %B4 : WORD;
	        Signals_3 AT %B6 : WORD;
	        Signals_4 AT %B8 : WORD;
	        Signals_5 AT %B10 : WORD;
	        Signals_6 AT %B12 : WORD;
	        Signals_7 AT %B14 : WORD;
	        Signals_8 AT %B16 : WORD;
	        Signals_9 AT %B18 : WORD;
	    END_STRUCT;
	END_TYPE

	TYPE
        {S7.extern=ReadWrite}
        {#ix-attr:[Container(Layout.Wrap)]}
	    keyence_iv3_ToolResult_28_Input_Layout : STRUCT
	        Signals_0 AT %B0 : WORD;
	        Signals_1 AT %B2 : WORD;
	        Signals_2 AT %B4 : WORD;
	        Signals_3 AT %B6 : WORD;
	        Signals_4 AT %B8 : WORD;
	        Signals_5 AT %B10 : WORD;
	        Signals_6 AT %B12 : WORD;
	        Signals_7 AT %B14 : WORD;
	        Signals_8 AT %B16 : WORD;
	        Signals_9 AT %B18 : WORD;
	    END_STRUCT;
	END_TYPE

	TYPE
        {S7.extern=ReadWrite}
        {#ix-attr:[Container(Layout.Wrap)]}
	    keyence_iv3_ToolResult_29_Input_Layout : STRUCT
	        Signals_0 AT %B0 : WORD;
	        Signals_1 AT %B2 : WORD;
	        Signals_2 AT %B4 : WORD;
	        Signals_3 AT %B6 : WORD;
	        Signals_4 AT %B8 : WORD;
	        Signals_5 AT %B10 : WORD;
	        Signals_6 AT %B12 : WORD;
	        Signals_7 AT %B14 : WORD;
	        Signals_8 AT %B16 : WORD;
	        Signals_9 AT %B18 : WORD;
	    END_STRUCT;
	END_TYPE

	TYPE
        {S7.extern=ReadWrite}
        {#ix-attr:[Container(Layout.Wrap)]}
	    keyence_iv3_ToolResult_3_Input_Layout : STRUCT
	        Signals_0 AT %B0 : WORD;
	        Signals_1 AT %B2 : WORD;
	        Signals_2 AT %B4 : WORD;
	        Signals_3 AT %B6 : WORD;
	        Signals_4 AT %B8 : WORD;
	        Signals_5 AT %B10 : WORD;
	        Signals_6 AT %B12 : WORD;
	        Signals_7 AT %B14 : WORD;
	        Signals_8 AT %B16 : WORD;
	        Signals_9 AT %B18 : WORD;
	    END_STRUCT;
	END_TYPE

	TYPE
        {S7.extern=ReadWrite}
        {#ix-attr:[Container(Layout.Wrap)]}
	    keyence_iv3_ToolResult_30_Input_Layout : STRUCT
	        Signals_0 AT %B0 : WORD;
	        Signals_1 AT %B2 : WORD;
	        Signals_2 AT %B4 : WORD;
	        Signals_3 AT %B6 : WORD;
	        Signals_4 AT %B8 : WORD;
	        Signals_5 AT %B10 : WORD;
	        Signals_6 AT %B12 : WORD;
	        Signals_7 AT %B14 : WORD;
	        Signals_8 AT %B16 : WORD;
	        Signals_9 AT %B18 : WORD;
	    END_STRUCT;
	END_TYPE

	TYPE
        {S7.extern=ReadWrite}
        {#ix-attr:[Container(Layout.Wrap)]}
	    keyence_iv3_ToolResult_31_Input_Layout : STRUCT
	        Signals_0 AT %B0 : WORD;
	        Signals_1 AT %B2 : WORD;
	        Signals_2 AT %B4 : WORD;
	        Signals_3 AT %B6 : WORD;
	        Signals_4 AT %B8 : WORD;
	        Signals_5 AT %B10 : WORD;
	        Signals_6 AT %B12 : WORD;
	        Signals_7 AT %B14 : WORD;
	        Signals_8 AT %B16 : WORD;
	        Signals_9 AT %B18 : WORD;
	    END_STRUCT;
	END_TYPE

	TYPE
        {S7.extern=ReadWrite}
        {#ix-attr:[Container(Layout.Wrap)]}
	    keyence_iv3_ToolResult_32_Input_Layout : STRUCT
	        Signals_0 AT %B0 : WORD;
	        Signals_1 AT %B2 : WORD;
	        Signals_2 AT %B4 : WORD;
	        Signals_3 AT %B6 : WORD;
	        Signals_4 AT %B8 : WORD;
	        Signals_5 AT %B10 : WORD;
	        Signals_6 AT %B12 : WORD;
	        Signals_7 AT %B14 : WORD;
	        Signals_8 AT %B16 : WORD;
	        Signals_9 AT %B18 : WORD;
	    END_STRUCT;
	END_TYPE

	TYPE
        {S7.extern=ReadWrite}
        {#ix-attr:[Container(Layout.Wrap)]}
	    keyence_iv3_ToolResult_33_Input_Layout : STRUCT
	        Signals_0 AT %B0 : WORD;
	        Signals_1 AT %B2 : WORD;
	        Signals_2 AT %B4 : WORD;
	        Signals_3 AT %B6 : WORD;
	        Signals_4 AT %B8 : WORD;
	        Signals_5 AT %B10 : WORD;
	        Signals_6 AT %B12 : WORD;
	        Signals_7 AT %B14 : WORD;
	        Signals_8 AT %B16 : WORD;
	        Signals_9 AT %B18 : WORD;
	    END_STRUCT;
	END_TYPE

	TYPE
        {S7.extern=ReadWrite}
        {#ix-attr:[Container(Layout.Wrap)]}
	    keyence_iv3_ToolResult_34_Input_Layout : STRUCT
	        Signals_0 AT %B0 : WORD;
	        Signals_1 AT %B2 : WORD;
	        Signals_2 AT %B4 : WORD;
	        Signals_3 AT %B6 : WORD;
	        Signals_4 AT %B8 : WORD;
	        Signals_5 AT %B10 : WORD;
	        Signals_6 AT %B12 : WORD;
	        Signals_7 AT %B14 : WORD;
	        Signals_8 AT %B16 : WORD;
	        Signals_9 AT %B18 : WORD;
	    END_STRUCT;
	END_TYPE

	TYPE
        {S7.extern=ReadWrite}
        {#ix-attr:[Container(Layout.Wrap)]}
	    keyence_iv3_ToolResult_35_Input_Layout : STRUCT
	        Signals_0 AT %B0 : WORD;
	        Signals_1 AT %B2 : WORD;
	        Signals_2 AT %B4 : WORD;
	        Signals_3 AT %B6 : WORD;
	        Signals_4 AT %B8 : WORD;
	        Signals_5 AT %B10 : WORD;
	        Signals_6 AT %B12 : WORD;
	        Signals_7 AT %B14 : WORD;
	        Signals_8 AT %B16 : WORD;
	        Signals_9 AT %B18 : WORD;
	    END_STRUCT;
	END_TYPE

	TYPE
        {S7.extern=ReadWrite}
        {#ix-attr:[Container(Layout.Wrap)]}
	    keyence_iv3_ToolResult_36_Input_Layout : STRUCT
	        Signals_0 AT %B0 : WORD;
	        Signals_1 AT %B2 : WORD;
	        Signals_2 AT %B4 : WORD;
	        Signals_3 AT %B6 : WORD;
	        Signals_4 AT %B8 : WORD;
	        Signals_5 AT %B10 : WORD;
	        Signals_6 AT %B12 : WORD;
	        Signals_7 AT %B14 : WORD;
	        Signals_8 AT %B16 : WORD;
	        Signals_9 AT %B18 : WORD;
	    END_STRUCT;
	END_TYPE

	TYPE
        {S7.extern=ReadWrite}
        {#ix-attr:[Container(Layout.Wrap)]}
	    keyence_iv3_ToolResult_37_Input_Layout : STRUCT
	        Signals_0 AT %B0 : WORD;
	        Signals_1 AT %B2 : WORD;
	        Signals_2 AT %B4 : WORD;
	        Signals_3 AT %B6 : WORD;
	        Signals_4 AT %B8 : WORD;
	        Signals_5 AT %B10 : WORD;
	        Signals_6 AT %B12 : WORD;
	        Signals_7 AT %B14 : WORD;
	        Signals_8 AT %B16 : WORD;
	        Signals_9 AT %B18 : WORD;
	    END_STRUCT;
	END_TYPE

	TYPE
        {S7.extern=ReadWrite}
        {#ix-attr:[Container(Layout.Wrap)]}
	    keyence_iv3_ToolResult_38_Input_Layout : STRUCT
	        Signals_0 AT %B0 : WORD;
	        Signals_1 AT %B2 : WORD;
	        Signals_2 AT %B4 : WORD;
	        Signals_3 AT %B6 : WORD;
	        Signals_4 AT %B8 : WORD;
	        Signals_5 AT %B10 : WORD;
	        Signals_6 AT %B12 : WORD;
	        Signals_7 AT %B14 : WORD;
	        Signals_8 AT %B16 : WORD;
	        Signals_9 AT %B18 : WORD;
	    END_STRUCT;
	END_TYPE

	TYPE
        {S7.extern=ReadWrite}
        {#ix-attr:[Container(Layout.Wrap)]}
	    keyence_iv3_ToolResult_39_Input_Layout : STRUCT
	        Signals_0 AT %B0 : WORD;
	        Signals_1 AT %B2 : WORD;
	        Signals_2 AT %B4 : WORD;
	        Signals_3 AT %B6 : WORD;
	        Signals_4 AT %B8 : WORD;
	        Signals_5 AT %B10 : WORD;
	        Signals_6 AT %B12 : WORD;
	        Signals_7 AT %B14 : WORD;
	        Signals_8 AT %B16 : WORD;
	        Signals_9 AT %B18 : WORD;
	    END_STRUCT;
	END_TYPE

	TYPE
        {S7.extern=ReadWrite}
        {#ix-attr:[Container(Layout.Wrap)]}
	    keyence_iv3_ToolResult_4_Input_Layout : STRUCT
	        Signals_0 AT %B0 : WORD;
	        Signals_1 AT %B2 : WORD;
	        Signals_2 AT %B4 : WORD;
	        Signals_3 AT %B6 : WORD;
	        Signals_4 AT %B8 : WORD;
	        Signals_5 AT %B10 : WORD;
	        Signals_6 AT %B12 : WORD;
	        Signals_7 AT %B14 : WORD;
	        Signals_8 AT %B16 : WORD;
	        Signals_9 AT %B18 : WORD;
	    END_STRUCT;
	END_TYPE

	TYPE
        {S7.extern=ReadWrite}
        {#ix-attr:[Container(Layout.Wrap)]}
	    keyence_iv3_ToolResult_40_Input_Layout : STRUCT
	        Signals_0 AT %B0 : WORD;
	        Signals_1 AT %B2 : WORD;
	        Signals_2 AT %B4 : WORD;
	        Signals_3 AT %B6 : WORD;
	        Signals_4 AT %B8 : WORD;
	        Signals_5 AT %B10 : WORD;
	        Signals_6 AT %B12 : WORD;
	        Signals_7 AT %B14 : WORD;
	        Signals_8 AT %B16 : WORD;
	        Signals_9 AT %B18 : WORD;
	    END_STRUCT;
	END_TYPE

	TYPE
        {S7.extern=ReadWrite}
        {#ix-attr:[Container(Layout.Wrap)]}
	    keyence_iv3_ToolResult_41_Input_Layout : STRUCT
	        Signals_0 AT %B0 : WORD;
	        Signals_1 AT %B2 : WORD;
	        Signals_2 AT %B4 : WORD;
	        Signals_3 AT %B6 : WORD;
	        Signals_4 AT %B8 : WORD;
	        Signals_5 AT %B10 : WORD;
	        Signals_6 AT %B12 : WORD;
	        Signals_7 AT %B14 : WORD;
	        Signals_8 AT %B16 : WORD;
	        Signals_9 AT %B18 : WORD;
	    END_STRUCT;
	END_TYPE

	TYPE
        {S7.extern=ReadWrite}
        {#ix-attr:[Container(Layout.Wrap)]}
	    keyence_iv3_ToolResult_42_Input_Layout : STRUCT
	        Signals_0 AT %B0 : WORD;
	        Signals_1 AT %B2 : WORD;
	        Signals_2 AT %B4 : WORD;
	        Signals_3 AT %B6 : WORD;
	        Signals_4 AT %B8 : WORD;
	        Signals_5 AT %B10 : WORD;
	        Signals_6 AT %B12 : WORD;
	        Signals_7 AT %B14 : WORD;
	        Signals_8 AT %B16 : WORD;
	        Signals_9 AT %B18 : WORD;
	    END_STRUCT;
	END_TYPE

	TYPE
        {S7.extern=ReadWrite}
        {#ix-attr:[Container(Layout.Wrap)]}
	    keyence_iv3_ToolResult_43_Input_Layout : STRUCT
	        Signals_0 AT %B0 : WORD;
	        Signals_1 AT %B2 : WORD;
	        Signals_2 AT %B4 : WORD;
	        Signals_3 AT %B6 : WORD;
	        Signals_4 AT %B8 : WORD;
	        Signals_5 AT %B10 : WORD;
	        Signals_6 AT %B12 : WORD;
	        Signals_7 AT %B14 : WORD;
	        Signals_8 AT %B16 : WORD;
	        Signals_9 AT %B18 : WORD;
	    END_STRUCT;
	END_TYPE

	TYPE
        {S7.extern=ReadWrite}
        {#ix-attr:[Container(Layout.Wrap)]}
	    keyence_iv3_ToolResult_44_Input_Layout : STRUCT
	        Signals_0 AT %B0 : WORD;
	        Signals_1 AT %B2 : WORD;
	        Signals_2 AT %B4 : WORD;
	        Signals_3 AT %B6 : WORD;
	        Signals_4 AT %B8 : WORD;
	        Signals_5 AT %B10 : WORD;
	        Signals_6 AT %B12 : WORD;
	        Signals_7 AT %B14 : WORD;
	        Signals_8 AT %B16 : WORD;
	        Signals_9 AT %B18 : WORD;
	    END_STRUCT;
	END_TYPE

	TYPE
        {S7.extern=ReadWrite}
        {#ix-attr:[Container(Layout.Wrap)]}
	    keyence_iv3_ToolResult_45_Input_Layout : STRUCT
	        Signals_0 AT %B0 : WORD;
	        Signals_1 AT %B2 : WORD;
	        Signals_2 AT %B4 : WORD;
	        Signals_3 AT %B6 : WORD;
	        Signals_4 AT %B8 : WORD;
	        Signals_5 AT %B10 : WORD;
	        Signals_6 AT %B12 : WORD;
	        Signals_7 AT %B14 : WORD;
	        Signals_8 AT %B16 : WORD;
	        Signals_9 AT %B18 : WORD;
	    END_STRUCT;
	END_TYPE

	TYPE
        {S7.extern=ReadWrite}
        {#ix-attr:[Container(Layout.Wrap)]}
	    keyence_iv3_ToolResult_46_Input_Layout : STRUCT
	        Signals_0 AT %B0 : WORD;
	        Signals_1 AT %B2 : WORD;
	        Signals_2 AT %B4 : WORD;
	        Signals_3 AT %B6 : WORD;
	        Signals_4 AT %B8 : WORD;
	        Signals_5 AT %B10 : WORD;
	        Signals_6 AT %B12 : WORD;
	        Signals_7 AT %B14 : WORD;
	        Signals_8 AT %B16 : WORD;
	        Signals_9 AT %B18 : WORD;
	    END_STRUCT;
	END_TYPE

	TYPE
        {S7.extern=ReadWrite}
        {#ix-attr:[Container(Layout.Wrap)]}
	    keyence_iv3_ToolResult_47_Input_Layout : STRUCT
	        Signals_0 AT %B0 : WORD;
	        Signals_1 AT %B2 : WORD;
	        Signals_2 AT %B4 : WORD;
	        Signals_3 AT %B6 : WORD;
	        Signals_4 AT %B8 : WORD;
	        Signals_5 AT %B10 : WORD;
	        Signals_6 AT %B12 : WORD;
	        Signals_7 AT %B14 : WORD;
	        Signals_8 AT %B16 : WORD;
	        Signals_9 AT %B18 : WORD;
	    END_STRUCT;
	END_TYPE

	TYPE
        {S7.extern=ReadWrite}
        {#ix-attr:[Container(Layout.Wrap)]}
	    keyence_iv3_ToolResult_48_Input_Layout : STRUCT
	        Signals_0 AT %B0 : WORD;
	        Signals_1 AT %B2 : WORD;
	        Signals_2 AT %B4 : WORD;
	        Signals_3 AT %B6 : WORD;
	        Signals_4 AT %B8 : WORD;
	        Signals_5 AT %B10 : WORD;
	        Signals_6 AT %B12 : WORD;
	        Signals_7 AT %B14 : WORD;
	        Signals_8 AT %B16 : WORD;
	        Signals_9 AT %B18 : WORD;
	    END_STRUCT;
	END_TYPE

	TYPE
        {S7.extern=ReadWrite}
        {#ix-attr:[Container(Layout.Wrap)]}
	    keyence_iv3_ToolResult_49_Input_Layout : STRUCT
	        Signals_0 AT %B0 : WORD;
	        Signals_1 AT %B2 : WORD;
	        Signals_2 AT %B4 : WORD;
	        Signals_3 AT %B6 : WORD;
	        Signals_4 AT %B8 : WORD;
	        Signals_5 AT %B10 : WORD;
	        Signals_6 AT %B12 : WORD;
	        Signals_7 AT %B14 : WORD;
	        Signals_8 AT %B16 : WORD;
	        Signals_9 AT %B18 : WORD;
	    END_STRUCT;
	END_TYPE

	TYPE
        {S7.extern=ReadWrite}
        {#ix-attr:[Container(Layout.Wrap)]}
	    keyence_iv3_ToolResult_5_Input_Layout : STRUCT
	        Signals_0 AT %B0 : WORD;
	        Signals_1 AT %B2 : WORD;
	        Signals_2 AT %B4 : WORD;
	        Signals_3 AT %B6 : WORD;
	        Signals_4 AT %B8 : WORD;
	        Signals_5 AT %B10 : WORD;
	        Signals_6 AT %B12 : WORD;
	        Signals_7 AT %B14 : WORD;
	        Signals_8 AT %B16 : WORD;
	        Signals_9 AT %B18 : WORD;
	    END_STRUCT;
	END_TYPE

	TYPE
        {S7.extern=ReadWrite}
        {#ix-attr:[Container(Layout.Wrap)]}
	    keyence_iv3_ToolResult_50_Input_Layout : STRUCT
	        Signals_0 AT %B0 : WORD;
	        Signals_1 AT %B2 : WORD;
	        Signals_2 AT %B4 : WORD;
	        Signals_3 AT %B6 : WORD;
	        Signals_4 AT %B8 : WORD;
	        Signals_5 AT %B10 : WORD;
	        Signals_6 AT %B12 : WORD;
	        Signals_7 AT %B14 : WORD;
	        Signals_8 AT %B16 : WORD;
	        Signals_9 AT %B18 : WORD;
	    END_STRUCT;
	END_TYPE

	TYPE
        {S7.extern=ReadWrite}
        {#ix-attr:[Container(Layout.Wrap)]}
	    keyence_iv3_ToolResult_51_Input_Layout : STRUCT
	        Signals_0 AT %B0 : WORD;
	        Signals_1 AT %B2 : WORD;
	        Signals_2 AT %B4 : WORD;
	        Signals_3 AT %B6 : WORD;
	        Signals_4 AT %B8 : WORD;
	        Signals_5 AT %B10 : WORD;
	        Signals_6 AT %B12 : WORD;
	        Signals_7 AT %B14 : WORD;
	        Signals_8 AT %B16 : WORD;
	        Signals_9 AT %B18 : WORD;
	    END_STRUCT;
	END_TYPE

	TYPE
        {S7.extern=ReadWrite}
        {#ix-attr:[Container(Layout.Wrap)]}
	    keyence_iv3_ToolResult_52_Input_Layout : STRUCT
	        Signals_0 AT %B0 : WORD;
	        Signals_1 AT %B2 : WORD;
	        Signals_2 AT %B4 : WORD;
	        Signals_3 AT %B6 : WORD;
	        Signals_4 AT %B8 : WORD;
	        Signals_5 AT %B10 : WORD;
	        Signals_6 AT %B12 : WORD;
	        Signals_7 AT %B14 : WORD;
	        Signals_8 AT %B16 : WORD;
	        Signals_9 AT %B18 : WORD;
	    END_STRUCT;
	END_TYPE

	TYPE
        {S7.extern=ReadWrite}
        {#ix-attr:[Container(Layout.Wrap)]}
	    keyence_iv3_ToolResult_53_Input_Layout : STRUCT
	        Signals_0 AT %B0 : WORD;
	        Signals_1 AT %B2 : WORD;
	        Signals_2 AT %B4 : WORD;
	        Signals_3 AT %B6 : WORD;
	        Signals_4 AT %B8 : WORD;
	        Signals_5 AT %B10 : WORD;
	        Signals_6 AT %B12 : WORD;
	        Signals_7 AT %B14 : WORD;
	        Signals_8 AT %B16 : WORD;
	        Signals_9 AT %B18 : WORD;
	    END_STRUCT;
	END_TYPE

	TYPE
        {S7.extern=ReadWrite}
        {#ix-attr:[Container(Layout.Wrap)]}
	    keyence_iv3_ToolResult_54_Input_Layout : STRUCT
	        Signals_0 AT %B0 : WORD;
	        Signals_1 AT %B2 : WORD;
	        Signals_2 AT %B4 : WORD;
	        Signals_3 AT %B6 : WORD;
	        Signals_4 AT %B8 : WORD;
	        Signals_5 AT %B10 : WORD;
	        Signals_6 AT %B12 : WORD;
	        Signals_7 AT %B14 : WORD;
	        Signals_8 AT %B16 : WORD;
	        Signals_9 AT %B18 : WORD;
	    END_STRUCT;
	END_TYPE

	TYPE
        {S7.extern=ReadWrite}
        {#ix-attr:[Container(Layout.Wrap)]}
	    keyence_iv3_ToolResult_55_Input_Layout : STRUCT
	        Signals_0 AT %B0 : WORD;
	        Signals_1 AT %B2 : WORD;
	        Signals_2 AT %B4 : WORD;
	        Signals_3 AT %B6 : WORD;
	        Signals_4 AT %B8 : WORD;
	        Signals_5 AT %B10 : WORD;
	        Signals_6 AT %B12 : WORD;
	        Signals_7 AT %B14 : WORD;
	        Signals_8 AT %B16 : WORD;
	        Signals_9 AT %B18 : WORD;
	    END_STRUCT;
	END_TYPE

	TYPE
        {S7.extern=ReadWrite}
        {#ix-attr:[Container(Layout.Wrap)]}
	    keyence_iv3_ToolResult_56_Input_Layout : STRUCT
	        Signals_0 AT %B0 : WORD;
	        Signals_1 AT %B2 : WORD;
	        Signals_2 AT %B4 : WORD;
	        Signals_3 AT %B6 : WORD;
	        Signals_4 AT %B8 : WORD;
	        Signals_5 AT %B10 : WORD;
	        Signals_6 AT %B12 : WORD;
	        Signals_7 AT %B14 : WORD;
	        Signals_8 AT %B16 : WORD;
	        Signals_9 AT %B18 : WORD;
	    END_STRUCT;
	END_TYPE

	TYPE
        {S7.extern=ReadWrite}
        {#ix-attr:[Container(Layout.Wrap)]}
	    keyence_iv3_ToolResult_57_Input_Layout : STRUCT
	        Signals_0 AT %B0 : WORD;
	        Signals_1 AT %B2 : WORD;
	        Signals_2 AT %B4 : WORD;
	        Signals_3 AT %B6 : WORD;
	        Signals_4 AT %B8 : WORD;
	        Signals_5 AT %B10 : WORD;
	        Signals_6 AT %B12 : WORD;
	        Signals_7 AT %B14 : WORD;
	        Signals_8 AT %B16 : WORD;
	        Signals_9 AT %B18 : WORD;
	    END_STRUCT;
	END_TYPE

	TYPE
        {S7.extern=ReadWrite}
        {#ix-attr:[Container(Layout.Wrap)]}
	    keyence_iv3_ToolResult_58_Input_Layout : STRUCT
	        Signals_0 AT %B0 : WORD;
	        Signals_1 AT %B2 : WORD;
	        Signals_2 AT %B4 : WORD;
	        Signals_3 AT %B6 : WORD;
	        Signals_4 AT %B8 : WORD;
	        Signals_5 AT %B10 : WORD;
	        Signals_6 AT %B12 : WORD;
	        Signals_7 AT %B14 : WORD;
	        Signals_8 AT %B16 : WORD;
	        Signals_9 AT %B18 : WORD;
	    END_STRUCT;
	END_TYPE

	TYPE
        {S7.extern=ReadWrite}
        {#ix-attr:[Container(Layout.Wrap)]}
	    keyence_iv3_ToolResult_59_Input_Layout : STRUCT
	        Signals_0 AT %B0 : WORD;
	        Signals_1 AT %B2 : WORD;
	        Signals_2 AT %B4 : WORD;
	        Signals_3 AT %B6 : WORD;
	        Signals_4 AT %B8 : WORD;
	        Signals_5 AT %B10 : WORD;
	        Signals_6 AT %B12 : WORD;
	        Signals_7 AT %B14 : WORD;
	        Signals_8 AT %B16 : WORD;
	        Signals_9 AT %B18 : WORD;
	    END_STRUCT;
	END_TYPE

	TYPE
        {S7.extern=ReadWrite}
        {#ix-attr:[Container(Layout.Wrap)]}
	    keyence_iv3_ToolResult_6_Input_Layout : STRUCT
	        Signals_0 AT %B0 : WORD;
	        Signals_1 AT %B2 : WORD;
	        Signals_2 AT %B4 : WORD;
	        Signals_3 AT %B6 : WORD;
	        Signals_4 AT %B8 : WORD;
	        Signals_5 AT %B10 : WORD;
	        Signals_6 AT %B12 : WORD;
	        Signals_7 AT %B14 : WORD;
	        Signals_8 AT %B16 : WORD;
	        Signals_9 AT %B18 : WORD;
	    END_STRUCT;
	END_TYPE

	TYPE
        {S7.extern=ReadWrite}
        {#ix-attr:[Container(Layout.Wrap)]}
	    keyence_iv3_ToolResult_60_Input_Layout : STRUCT
	        Signals_0 AT %B0 : WORD;
	        Signals_1 AT %B2 : WORD;
	        Signals_2 AT %B4 : WORD;
	        Signals_3 AT %B6 : WORD;
	        Signals_4 AT %B8 : WORD;
	        Signals_5 AT %B10 : WORD;
	        Signals_6 AT %B12 : WORD;
	        Signals_7 AT %B14 : WORD;
	        Signals_8 AT %B16 : WORD;
	        Signals_9 AT %B18 : WORD;
	    END_STRUCT;
	END_TYPE

	TYPE
        {S7.extern=ReadWrite}
        {#ix-attr:[Container(Layout.Wrap)]}
	    keyence_iv3_ToolResult_61_Input_Layout : STRUCT
	        Signals_0 AT %B0 : WORD;
	        Signals_1 AT %B2 : WORD;
	        Signals_2 AT %B4 : WORD;
	        Signals_3 AT %B6 : WORD;
	        Signals_4 AT %B8 : WORD;
	        Signals_5 AT %B10 : WORD;
	        Signals_6 AT %B12 : WORD;
	        Signals_7 AT %B14 : WORD;
	        Signals_8 AT %B16 : WORD;
	        Signals_9 AT %B18 : WORD;
	    END_STRUCT;
	END_TYPE

	TYPE
        {S7.extern=ReadWrite}
        {#ix-attr:[Container(Layout.Wrap)]}
	    keyence_iv3_ToolResult_62_Input_Layout : STRUCT
	        Signals_0 AT %B0 : WORD;
	        Signals_1 AT %B2 : WORD;
	        Signals_2 AT %B4 : WORD;
	        Signals_3 AT %B6 : WORD;
	        Signals_4 AT %B8 : WORD;
	        Signals_5 AT %B10 : WORD;
	        Signals_6 AT %B12 : WORD;
	        Signals_7 AT %B14 : WORD;
	        Signals_8 AT %B16 : WORD;
	        Signals_9 AT %B18 : WORD;
	    END_STRUCT;
	END_TYPE

	TYPE
        {S7.extern=ReadWrite}
        {#ix-attr:[Container(Layout.Wrap)]}
	    keyence_iv3_ToolResult_63_Input_Layout : STRUCT
	        Signals_0 AT %B0 : WORD;
	        Signals_1 AT %B2 : WORD;
	        Signals_2 AT %B4 : WORD;
	        Signals_3 AT %B6 : WORD;
	        Signals_4 AT %B8 : WORD;
	        Signals_5 AT %B10 : WORD;
	        Signals_6 AT %B12 : WORD;
	        Signals_7 AT %B14 : WORD;
	        Signals_8 AT %B16 : WORD;
	        Signals_9 AT %B18 : WORD;
	    END_STRUCT;
	END_TYPE

	TYPE
        {S7.extern=ReadWrite}
        {#ix-attr:[Container(Layout.Wrap)]}
	    keyence_iv3_ToolResult_64_Input_Layout : STRUCT
	        Signals_0 AT %B0 : WORD;
	        Signals_1 AT %B2 : WORD;
	        Signals_2 AT %B4 : WORD;
	        Signals_3 AT %B6 : WORD;
	        Signals_4 AT %B8 : WORD;
	        Signals_5 AT %B10 : WORD;
	        Signals_6 AT %B12 : WORD;
	        Signals_7 AT %B14 : WORD;
	        Signals_8 AT %B16 : WORD;
	        Signals_9 AT %B18 : WORD;
	    END_STRUCT;
	END_TYPE

	TYPE
        {S7.extern=ReadWrite}
        {#ix-attr:[Container(Layout.Wrap)]}
	    keyence_iv3_ToolResult_7_Input_Layout : STRUCT
	        Signals_0 AT %B0 : WORD;
	        Signals_1 AT %B2 : WORD;
	        Signals_2 AT %B4 : WORD;
	        Signals_3 AT %B6 : WORD;
	        Signals_4 AT %B8 : WORD;
	        Signals_5 AT %B10 : WORD;
	        Signals_6 AT %B12 : WORD;
	        Signals_7 AT %B14 : WORD;
	        Signals_8 AT %B16 : WORD;
	        Signals_9 AT %B18 : WORD;
	    END_STRUCT;
	END_TYPE

	TYPE
        {S7.extern=ReadWrite}
        {#ix-attr:[Container(Layout.Wrap)]}
	    keyence_iv3_ToolResult_8_Input_Layout : STRUCT
	        Signals_0 AT %B0 : WORD;
	        Signals_1 AT %B2 : WORD;
	        Signals_2 AT %B4 : WORD;
	        Signals_3 AT %B6 : WORD;
	        Signals_4 AT %B8 : WORD;
	        Signals_5 AT %B10 : WORD;
	        Signals_6 AT %B12 : WORD;
	        Signals_7 AT %B14 : WORD;
	        Signals_8 AT %B16 : WORD;
	        Signals_9 AT %B18 : WORD;
	    END_STRUCT;
	END_TYPE

	TYPE
        {S7.extern=ReadWrite}
        {#ix-attr:[Container(Layout.Wrap)]}
	    keyence_iv3_ToolResult_9_Input_Layout : STRUCT
	        Signals_0 AT %B0 : WORD;
	        Signals_1 AT %B2 : WORD;
	        Signals_2 AT %B4 : WORD;
	        Signals_3 AT %B6 : WORD;
	        Signals_4 AT %B8 : WORD;
	        Signals_5 AT %B10 : WORD;
	        Signals_6 AT %B12 : WORD;
	        Signals_7 AT %B14 : WORD;
	        Signals_8 AT %B16 : WORD;
	        Signals_9 AT %B18 : WORD;
	    END_STRUCT;
	END_TYPE

	TYPE
        {S7.extern=ReadWrite}
        {#ix-attr:[Container(Layout.Wrap)]}
	    keyence_sr_1000_BusyStatus_Input_Layout : STRUCT
	        Signals_0 AT %X0.0 : BOOL;
	        Signals_1 AT %X0.1 : BOOL;
	        Signals_2 AT %X0.2 : BOOL;
	        Signals_3 AT %X0.3 : BOOL;
	        Signals_4 AT %X0.4 : BOOL;
	    END_STRUCT;
	END_TYPE

	TYPE
        {S7.extern=ReadWrite}
        {#ix-attr:[Container(Layout.Wrap)]}
	    keyence_sr_1000_CompletionClearControl_Output_Layout : STRUCT
	        Signals_0 AT %X0.0 : BOOL;
	        Signals_1 AT %X0.1 : BOOL;
	        Signals_2 AT %X0.2 : BOOL;
	        Signals_3 AT %X0.3 : BOOL;
	        Signals_4 AT %X0.7 : BOOL;
	    END_STRUCT;
	END_TYPE

	TYPE
        {S7.extern=ReadWrite}
        {#ix-attr:[Container(Layout.Wrap)]}
	    keyence_sr_1000_CompletionStatus_Input_Layout : STRUCT
	        Signals_0 AT %X0.0 : BOOL;
	        Signals_1 AT %X0.1 : BOOL;
	        Signals_2 AT %X0.2 : BOOL;
	        Signals_3 AT %X0.3 : BOOL;
	        Signals_4 AT %X0.7 : BOOL;
	    END_STRUCT;
	END_TYPE

	TYPE
        {S7.extern=ReadWrite}
        {#ix-attr:[Container(Layout.Wrap)]}
	    keyence_sr_1000_ErrorStatus_Input_Layout : STRUCT
	        Signals_0 AT %X0.0 : BOOL;
	        Signals_1 AT %X0.1 : BOOL;
	        Signals_2 AT %X0.2 : BOOL;
	        Signals_3 AT %X0.3 : BOOL;
	        Signals_4 AT %X0.7 : BOOL;
	    END_STRUCT;
	END_TYPE

	TYPE
        {S7.extern=ReadWrite}
        {#ix-attr:[Container(Layout.Wrap)]}
	    keyence_sr_1000_HandshakeAndGeneralErrorStatus_Input_Layout : STRUCT
	        Signals_0 AT %X0.0 : BOOL;
	        Signals_1 AT %X0.1 : BOOL;
	        Signals_2 AT %X0.2 : BOOL;
	        Signals_3 AT %X0.6 : BOOL;
	        Signals_4 AT %X0.7 : BOOL;
	    END_STRUCT;
	END_TYPE

	TYPE
        {S7.extern=ReadWrite}
        {#ix-attr:[Container(Layout.Wrap)]}
	    keyence_sr_1000_LatchAndErrorClearControl_Output_Layout : STRUCT
	        Signals_0 AT %X0.1 : BOOL;
	        Signals_1 AT %X0.7 : BOOL;
	    END_STRUCT;
	END_TYPE

	TYPE
        {S7.extern=ReadWrite}
        {#ix-attr:[Container(Layout.Wrap)]}
	    keyence_sr_1000_MatchingLevelAndTotalEvaluationGradeStatus_Input_Layout : STRUCT
	        Signals_0 AT %B0 : WORD;
	        Signals_1 AT %B2 : WORD;
	        Signals_2 AT %B4 : WORD;
	        Signals_3 AT %B6 : WORD;
	    END_STRUCT;
	END_TYPE

	TYPE
        {S7.extern=ReadWrite}
        {#ix-attr:[Container(Layout.Wrap)]}
	    keyence_sr_1000_OperationInstructionControl_Output_Layout : STRUCT
	        Signals_0 AT %X0.0 : BOOL;
	        Signals_1 AT %X0.1 : BOOL;
	        Signals_2 AT %X0.2 : BOOL;
	        Signals_3 AT %X0.3 : BOOL;
	    END_STRUCT;
	END_TYPE

	TYPE
        {S7.extern=ReadWrite}
        {#ix-attr:[Container(Layout.Wrap)]}
	    keyence_sr_1000_OperationResultStatus_Input_Layout : STRUCT
	        Signals_0 AT %B0 : WORD;
	        Signals_1 AT %B2 : WORD;
	        Signals_2 AT %B4 : WORD;
	        Signals_3 AT %B6 : WORD;
	        Signals_4 AT %B8 : WORD;
	        Signals_5 AT %B10 : WORD;
	        Signals_6 AT %B12 : WORD;
	        Signals_7 AT %B14 : WORD;
	        Signals_8 AT %B16 : WORD;
	        Signals_9 AT %B18 : WORD;
	    END_STRUCT;
	END_TYPE

	TYPE
        {S7.extern=ReadWrite}
        {#ix-attr:[Container(Layout.Wrap)]}
	    keyence_sr_1000_ParameterBank_Output_Layout : STRUCT
	        Signals_0 AT %B0 : WORD;
	    END_STRUCT;
	END_TYPE

	TYPE
        {S7.extern=ReadWrite}
        {#ix-attr:[Container(Layout.Wrap)]}
	    keyence_sr_1000_ResultData_128_Input_Layout : STRUCT
	        Signals_0 AT %B0 : WORD;
	        Signals_1 AT %B2 : WORD;
	        Signals_2 AT %B4 : WORD;
	        Signals_3 AT %B6 : WORD;
	        Signals_4 AT %B8 : ARRAY[0..127] OF BYTE;
	    END_STRUCT;
	END_TYPE

	TYPE
        {S7.extern=ReadWrite}
        {#ix-attr:[Container(Layout.Wrap)]}
	    keyence_sr_1000_TerminalStatus_Input_Layout : STRUCT
	        Signals_0 AT %X0.0 : BOOL;
	        Signals_1 AT %X0.1 : BOOL;
	        Signals_2 AT %X0.4 : BOOL;
	        Signals_3 AT %X0.5 : BOOL;
	        Signals_4 AT %X0.6 : BOOL;
	    END_STRUCT;
	END_TYPE

	TYPE
        {S7.extern=ReadWrite}
        {#ix-attr:[Container(Layout.Wrap)]}
	    keyence_sr_1000_UnstableReadStatus_Input_Layout : STRUCT
	        Signals_0 AT %X0.0 : BOOL;
	        Signals_1 AT %X0.1 : BOOL;
	        Signals_2 AT %X0.2 : BOOL;
	        Signals_3 AT %X0.3 : BOOL;
	        Signals_4 AT %X0.4 : BOOL;
	    END_STRUCT;
	END_TYPE

	TYPE
        {S7.extern=ReadWrite}
        {#ix-attr:[Container(Layout.Wrap)]}
	    keyence_sr_1000_UserData_128_Output_Layout : STRUCT
	        Signals_0 AT %B0 : WORD;
	        Signals_1 AT %B2 : ARRAY[0..127] OF BYTE;
	    END_STRUCT;
	END_TYPE

	TYPE
        {S7.extern=ReadWrite}
        {#ix-attr:[Container(Layout.Wrap)]}
	    keyence_sr_750_BusyStatus_Input_Layout : STRUCT
	        Signals_0 AT %X0.0 : BOOL;
	        Signals_1 AT %X0.1 : BOOL;
	        Signals_2 AT %X0.2 : BOOL;
	        Signals_3 AT %X0.3 : BOOL;
	        Signals_4 AT %X0.4 : BOOL;
	    END_STRUCT;
	END_TYPE

	TYPE
        {S7.extern=ReadWrite}
        {#ix-attr:[Container(Layout.Wrap)]}
	    keyence_sr_750_CompletionClearControl_Output_Layout : STRUCT
	        Signals_0 AT %X0.0 : BOOL;
	        Signals_1 AT %X0.1 : BOOL;
	        Signals_2 AT %X0.2 : BOOL;
	        Signals_3 AT %X0.3 : BOOL;
	        Signals_4 AT %X0.7 : BOOL;
	    END_STRUCT;
	END_TYPE

	TYPE
        {S7.extern=ReadWrite}
        {#ix-attr:[Container(Layout.Wrap)]}
	    keyence_sr_750_CompletionStatus_Input_Layout : STRUCT
	        Signals_0 AT %X0.0 : BOOL;
	        Signals_1 AT %X0.1 : BOOL;
	        Signals_2 AT %X0.2 : BOOL;
	        Signals_3 AT %X0.3 : BOOL;
	        Signals_4 AT %X0.7 : BOOL;
	    END_STRUCT;
	END_TYPE

	TYPE
        {S7.extern=ReadWrite}
        {#ix-attr:[Container(Layout.Wrap)]}
	    keyence_sr_750_ErrorStatus_Input_Layout : STRUCT
	        Signals_0 AT %X0.0 : BOOL;
	        Signals_1 AT %X0.1 : BOOL;
	        Signals_2 AT %X0.2 : BOOL;
	        Signals_3 AT %X0.3 : BOOL;
	        Signals_4 AT %X0.7 : BOOL;
	    END_STRUCT;
	END_TYPE

	TYPE
        {S7.extern=ReadWrite}
        {#ix-attr:[Container(Layout.Wrap)]}
	    keyence_sr_750_HandshakeAndGeneralErrorStatus_Input_Layout : STRUCT
	        Signals_0 AT %X0.0 : BOOL;
	        Signals_1 AT %X0.1 : BOOL;
	        Signals_2 AT %X0.2 : BOOL;
	        Signals_3 AT %X0.6 : BOOL;
	        Signals_4 AT %X0.7 : BOOL;
	    END_STRUCT;
	END_TYPE

	TYPE
        {S7.extern=ReadWrite}
        {#ix-attr:[Container(Layout.Wrap)]}
	    keyence_sr_750_LatchAndErrorClearControl_Output_Layout : STRUCT
	        Signals_0 AT %X0.1 : BOOL;
	        Signals_1 AT %X0.7 : BOOL;
	    END_STRUCT;
	END_TYPE

	TYPE
        {S7.extern=ReadWrite}
        {#ix-attr:[Container(Layout.Wrap)]}
	    keyence_sr_750_MatchingLevelAndTotalEvaluationGradeStatus_Input_Layout : STRUCT
	        Signals_0 AT %B0 : WORD;
	        Signals_1 AT %B2 : WORD;
	        Signals_2 AT %B4 : WORD;
	        Signals_3 AT %B6 : WORD;
	    END_STRUCT;
	END_TYPE

	TYPE
        {S7.extern=ReadWrite}
        {#ix-attr:[Container(Layout.Wrap)]}
	    keyence_sr_750_OperationInstructionControl_Output_Layout : STRUCT
	        Signals_0 AT %X0.0 : BOOL;
	        Signals_1 AT %X0.1 : BOOL;
	        Signals_2 AT %X0.2 : BOOL;
	        Signals_3 AT %X0.3 : BOOL;
	    END_STRUCT;
	END_TYPE

	TYPE
        {S7.extern=ReadWrite}
        {#ix-attr:[Container(Layout.Wrap)]}
	    keyence_sr_750_OperationResultStatus_Input_Layout : STRUCT
	        Signals_0 AT %B0 : WORD;
	        Signals_1 AT %B2 : WORD;
	        Signals_2 AT %B4 : WORD;
	        Signals_3 AT %B6 : WORD;
	        Signals_4 AT %B8 : WORD;
	        Signals_5 AT %B10 : WORD;
	        Signals_6 AT %B12 : WORD;
	        Signals_7 AT %B14 : WORD;
	        Signals_8 AT %B16 : WORD;
	        Signals_9 AT %B18 : WORD;
	    END_STRUCT;
	END_TYPE

	TYPE
        {S7.extern=ReadWrite}
        {#ix-attr:[Container(Layout.Wrap)]}
	    keyence_sr_750_ParameterBank_Output_Layout : STRUCT
	        Signals_0 AT %B0 : WORD;
	    END_STRUCT;
	END_TYPE

	TYPE
        {S7.extern=ReadWrite}
        {#ix-attr:[Container(Layout.Wrap)]}
	    keyence_sr_750_ResultData_128_Input_Layout : STRUCT
	        Signals_0 AT %B0 : WORD;
	        Signals_1 AT %B2 : WORD;
	        Signals_2 AT %B4 : WORD;
	        Signals_3 AT %B6 : WORD;
	        Signals_4 AT %B8 : ARRAY[0..127] OF BYTE;
	    END_STRUCT;
	END_TYPE

	TYPE
        {S7.extern=ReadWrite}
        {#ix-attr:[Container(Layout.Wrap)]}
	    keyence_sr_750_TerminalStatus_Input_Layout : STRUCT
	        Signals_0 AT %X0.0 : BOOL;
	        Signals_1 AT %X0.1 : BOOL;
	        Signals_2 AT %X0.4 : BOOL;
	        Signals_3 AT %X0.5 : BOOL;
	        Signals_4 AT %X0.6 : BOOL;
	    END_STRUCT;
	END_TYPE

	TYPE
        {S7.extern=ReadWrite}
        {#ix-attr:[Container(Layout.Wrap)]}
	    keyence_sr_750_UnstableReadStatus_Input_Layout : STRUCT
	        Signals_0 AT %X0.0 : BOOL;
	        Signals_1 AT %X0.1 : BOOL;
	        Signals_2 AT %X0.2 : BOOL;
	        Signals_3 AT %X0.3 : BOOL;
	        Signals_4 AT %X0.4 : BOOL;
	    END_STRUCT;
	END_TYPE

	TYPE
        {S7.extern=ReadWrite}
        {#ix-attr:[Container(Layout.Wrap)]}
	    keyence_sr_750_UserData_128_Output_Layout : STRUCT
	        Signals_0 AT %B0 : WORD;
	        Signals_1 AT %B2 : ARRAY[0..127] OF BYTE;
	    END_STRUCT;
	END_TYPE

	TYPE
        {S7.extern=ReadWrite}
        {#ix-attr:[Container(Layout.Wrap)]}
	    kuka_rb1_DIO512_Input_Layout : STRUCT
	        Signals_0_0 AT %X0.0 : BOOL;
	        Signals_0_1 AT %X0.1 : BOOL;
	        Signals_0_2 AT %X0.2 : BOOL;
	        Signals_0_3 AT %X0.3 : BOOL;
	        Signals_0_4 AT %X0.4 : BOOL;
	        Signals_0_5 AT %X0.5 : BOOL;
	        Signals_0_6 AT %X0.6 : BOOL;
	        Signals_0_7 AT %X0.7 : BOOL;
	        Signals_1_0 AT %X1.0 : BOOL;
	        Signals_1_1 AT %X1.1 : BOOL;
	        Signals_1_2 AT %X1.2 : BOOL;
	        Signals_1_3 AT %X1.3 : BOOL;
	        Signals_1_4 AT %X1.4 : BOOL;
	        Signals_1_5 AT %X1.5 : BOOL;
	        Signals_1_6 AT %X1.6 : BOOL;
	        Signals_1_7 AT %X1.7 : BOOL;
	        Signals_2_0 AT %X2.0 : BOOL;
	        Signals_2_1 AT %X2.1 : BOOL;
	        Signals_2_2 AT %X2.2 : BOOL;
	        Signals_2_3 AT %X2.3 : BOOL;
	        Signals_2_4 AT %X2.4 : BOOL;
	        Signals_2_5 AT %X2.5 : BOOL;
	        Signals_2_6 AT %X2.6 : BOOL;
	        Signals_2_7 AT %X2.7 : BOOL;
	        Signals_3_0 AT %X3.0 : BOOL;
	        Signals_3_1 AT %X3.1 : BOOL;
	        Signals_3_2 AT %X3.2 : BOOL;
	        Signals_3_3 AT %X3.3 : BOOL;
	        Signals_3_4 AT %X3.4 : BOOL;
	        Signals_3_5 AT %X3.5 : BOOL;
	        Signals_3_6 AT %X3.6 : BOOL;
	        Signals_3_7 AT %X3.7 : BOOL;
	        Signals_4_0 AT %X4.0 : BOOL;
	        Signals_4_1 AT %X4.1 : BOOL;
	        Signals_4_2 AT %X4.2 : BOOL;
	        Signals_4_3 AT %X4.3 : BOOL;
	        Signals_4_4 AT %X4.4 : BOOL;
	        Signals_4_5 AT %X4.5 : BOOL;
	        Signals_4_6 AT %X4.6 : BOOL;
	        Signals_4_7 AT %X4.7 : BOOL;
	        Signals_5_0 AT %X5.0 : BOOL;
	        Signals_5_1 AT %X5.1 : BOOL;
	        Signals_5_2 AT %X5.2 : BOOL;
	        Signals_5_3 AT %X5.3 : BOOL;
	        Signals_5_4 AT %X5.4 : BOOL;
	        Signals_5_5 AT %X5.5 : BOOL;
	        Signals_5_6 AT %X5.6 : BOOL;
	        Signals_5_7 AT %X5.7 : BOOL;
	        Signals_6_0 AT %X6.0 : BOOL;
	        Signals_6_1 AT %X6.1 : BOOL;
	        Signals_6_2 AT %X6.2 : BOOL;
	        Signals_6_3 AT %X6.3 : BOOL;
	        Signals_6_4 AT %X6.4 : BOOL;
	        Signals_6_5 AT %X6.5 : BOOL;
	        Signals_6_6 AT %X6.6 : BOOL;
	        Signals_6_7 AT %X6.7 : BOOL;
	        Signals_7_0 AT %X7.0 : BOOL;
	        Signals_7_1 AT %X7.1 : BOOL;
	        Signals_7_2 AT %X7.2 : BOOL;
	        Signals_7_3 AT %X7.3 : BOOL;
	        Signals_7_4 AT %X7.4 : BOOL;
	        Signals_7_5 AT %X7.5 : BOOL;
	        Signals_7_6 AT %X7.6 : BOOL;
	        Signals_7_7 AT %X7.7 : BOOL;
	        Signals_8_0 AT %X8.0 : BOOL;
	        Signals_8_1 AT %X8.1 : BOOL;
	        Signals_8_2 AT %X8.2 : BOOL;
	        Signals_8_3 AT %X8.3 : BOOL;
	        Signals_8_4 AT %X8.4 : BOOL;
	        Signals_8_5 AT %X8.5 : BOOL;
	        Signals_8_6 AT %X8.6 : BOOL;
	        Signals_8_7 AT %X8.7 : BOOL;
	        Signals_9_0 AT %X9.0 : BOOL;
	        Signals_9_1 AT %X9.1 : BOOL;
	        Signals_9_2 AT %X9.2 : BOOL;
	        Signals_9_3 AT %X9.3 : BOOL;
	        Signals_9_4 AT %X9.4 : BOOL;
	        Signals_9_5 AT %X9.5 : BOOL;
	        Signals_9_6 AT %X9.6 : BOOL;
	        Signals_9_7 AT %X9.7 : BOOL;
	        Signals_10_0 AT %X10.0 : BOOL;
	        Signals_10_1 AT %X10.1 : BOOL;
	        Signals_10_2 AT %X10.2 : BOOL;
	        Signals_10_3 AT %X10.3 : BOOL;
	        Signals_10_4 AT %X10.4 : BOOL;
	        Signals_10_5 AT %X10.5 : BOOL;
	        Signals_10_6 AT %X10.6 : BOOL;
	        Signals_10_7 AT %X10.7 : BOOL;
	        Signals_11_0 AT %X11.0 : BOOL;
	        Signals_11_1 AT %X11.1 : BOOL;
	        Signals_11_2 AT %X11.2 : BOOL;
	        Signals_11_3 AT %X11.3 : BOOL;
	        Signals_11_4 AT %X11.4 : BOOL;
	        Signals_11_5 AT %X11.5 : BOOL;
	        Signals_11_6 AT %X11.6 : BOOL;
	        Signals_11_7 AT %X11.7 : BOOL;
	        Signals_12_0 AT %X12.0 : BOOL;
	        Signals_12_1 AT %X12.1 : BOOL;
	        Signals_12_2 AT %X12.2 : BOOL;
	        Signals_12_3 AT %X12.3 : BOOL;
	        Signals_12_4 AT %X12.4 : BOOL;
	        Signals_12_5 AT %X12.5 : BOOL;
	        Signals_12_6 AT %X12.6 : BOOL;
	        Signals_12_7 AT %X12.7 : BOOL;
	        Signals_13_0 AT %X13.0 : BOOL;
	        Signals_13_1 AT %X13.1 : BOOL;
	        Signals_13_2 AT %X13.2 : BOOL;
	        Signals_13_3 AT %X13.3 : BOOL;
	        Signals_13_4 AT %X13.4 : BOOL;
	        Signals_13_5 AT %X13.5 : BOOL;
	        Signals_13_6 AT %X13.6 : BOOL;
	        Signals_13_7 AT %X13.7 : BOOL;
	        Signals_14_0 AT %X14.0 : BOOL;
	        Signals_14_1 AT %X14.1 : BOOL;
	        Signals_14_2 AT %X14.2 : BOOL;
	        Signals_14_3 AT %X14.3 : BOOL;
	        Signals_14_4 AT %X14.4 : BOOL;
	        Signals_14_5 AT %X14.5 : BOOL;
	        Signals_14_6 AT %X14.6 : BOOL;
	        Signals_14_7 AT %X14.7 : BOOL;
	        Signals_15_0 AT %X15.0 : BOOL;
	        Signals_15_1 AT %X15.1 : BOOL;
	        Signals_15_2 AT %X15.2 : BOOL;
	        Signals_15_3 AT %X15.3 : BOOL;
	        Signals_15_4 AT %X15.4 : BOOL;
	        Signals_15_5 AT %X15.5 : BOOL;
	        Signals_15_6 AT %X15.6 : BOOL;
	        Signals_15_7 AT %X15.7 : BOOL;
	        Signals_16_0 AT %X16.0 : BOOL;
	        Signals_16_1 AT %X16.1 : BOOL;
	        Signals_16_2 AT %X16.2 : BOOL;
	        Signals_16_3 AT %X16.3 : BOOL;
	        Signals_16_4 AT %X16.4 : BOOL;
	        Signals_16_5 AT %X16.5 : BOOL;
	        Signals_16_6 AT %X16.6 : BOOL;
	        Signals_16_7 AT %X16.7 : BOOL;
	        Signals_17_0 AT %X17.0 : BOOL;
	        Signals_17_1 AT %X17.1 : BOOL;
	        Signals_17_2 AT %X17.2 : BOOL;
	        Signals_17_3 AT %X17.3 : BOOL;
	        Signals_17_4 AT %X17.4 : BOOL;
	        Signals_17_5 AT %X17.5 : BOOL;
	        Signals_17_6 AT %X17.6 : BOOL;
	        Signals_17_7 AT %X17.7 : BOOL;
	        Signals_18_0 AT %X18.0 : BOOL;
	        Signals_18_1 AT %X18.1 : BOOL;
	        Signals_18_2 AT %X18.2 : BOOL;
	        Signals_18_3 AT %X18.3 : BOOL;
	        Signals_18_4 AT %X18.4 : BOOL;
	        Signals_18_5 AT %X18.5 : BOOL;
	        Signals_18_6 AT %X18.6 : BOOL;
	        Signals_18_7 AT %X18.7 : BOOL;
	        Signals_19_0 AT %X19.0 : BOOL;
	        Signals_19_1 AT %X19.1 : BOOL;
	        Signals_19_2 AT %X19.2 : BOOL;
	        Signals_19_3 AT %X19.3 : BOOL;
	        Signals_19_4 AT %X19.4 : BOOL;
	        Signals_19_5 AT %X19.5 : BOOL;
	        Signals_19_6 AT %X19.6 : BOOL;
	        Signals_19_7 AT %X19.7 : BOOL;
	        Signals_20_0 AT %X20.0 : BOOL;
	        Signals_20_1 AT %X20.1 : BOOL;
	        Signals_20_2 AT %X20.2 : BOOL;
	        Signals_20_3 AT %X20.3 : BOOL;
	        Signals_20_4 AT %X20.4 : BOOL;
	        Signals_20_5 AT %X20.5 : BOOL;
	        Signals_20_6 AT %X20.6 : BOOL;
	        Signals_20_7 AT %X20.7 : BOOL;
	        Signals_21_0 AT %X21.0 : BOOL;
	        Signals_21_1 AT %X21.1 : BOOL;
	        Signals_21_2 AT %X21.2 : BOOL;
	        Signals_21_3 AT %X21.3 : BOOL;
	        Signals_21_4 AT %X21.4 : BOOL;
	        Signals_21_5 AT %X21.5 : BOOL;
	        Signals_21_6 AT %X21.6 : BOOL;
	        Signals_21_7 AT %X21.7 : BOOL;
	        Signals_22_0 AT %X22.0 : BOOL;
	        Signals_22_1 AT %X22.1 : BOOL;
	        Signals_22_2 AT %X22.2 : BOOL;
	        Signals_22_3 AT %X22.3 : BOOL;
	        Signals_22_4 AT %X22.4 : BOOL;
	        Signals_22_5 AT %X22.5 : BOOL;
	        Signals_22_6 AT %X22.6 : BOOL;
	        Signals_22_7 AT %X22.7 : BOOL;
	        Signals_23_0 AT %X23.0 : BOOL;
	        Signals_23_1 AT %X23.1 : BOOL;
	        Signals_23_2 AT %X23.2 : BOOL;
	        Signals_23_3 AT %X23.3 : BOOL;
	        Signals_23_4 AT %X23.4 : BOOL;
	        Signals_23_5 AT %X23.5 : BOOL;
	        Signals_23_6 AT %X23.6 : BOOL;
	        Signals_23_7 AT %X23.7 : BOOL;
	        Signals_24_0 AT %X24.0 : BOOL;
	        Signals_24_1 AT %X24.1 : BOOL;
	        Signals_24_2 AT %X24.2 : BOOL;
	        Signals_24_3 AT %X24.3 : BOOL;
	        Signals_24_4 AT %X24.4 : BOOL;
	        Signals_24_5 AT %X24.5 : BOOL;
	        Signals_24_6 AT %X24.6 : BOOL;
	        Signals_24_7 AT %X24.7 : BOOL;
	        Signals_25_0 AT %X25.0 : BOOL;
	        Signals_25_1 AT %X25.1 : BOOL;
	        Signals_25_2 AT %X25.2 : BOOL;
	        Signals_25_3 AT %X25.3 : BOOL;
	        Signals_25_4 AT %X25.4 : BOOL;
	        Signals_25_5 AT %X25.5 : BOOL;
	        Signals_25_6 AT %X25.6 : BOOL;
	        Signals_25_7 AT %X25.7 : BOOL;
	        Signals_26_0 AT %X26.0 : BOOL;
	        Signals_26_1 AT %X26.1 : BOOL;
	        Signals_26_2 AT %X26.2 : BOOL;
	        Signals_26_3 AT %X26.3 : BOOL;
	        Signals_26_4 AT %X26.4 : BOOL;
	        Signals_26_5 AT %X26.5 : BOOL;
	        Signals_26_6 AT %X26.6 : BOOL;
	        Signals_26_7 AT %X26.7 : BOOL;
	        Signals_27_0 AT %X27.0 : BOOL;
	        Signals_27_1 AT %X27.1 : BOOL;
	        Signals_27_2 AT %X27.2 : BOOL;
	        Signals_27_3 AT %X27.3 : BOOL;
	        Signals_27_4 AT %X27.4 : BOOL;
	        Signals_27_5 AT %X27.5 : BOOL;
	        Signals_27_6 AT %X27.6 : BOOL;
	        Signals_27_7 AT %X27.7 : BOOL;
	        Signals_28_0 AT %X28.0 : BOOL;
	        Signals_28_1 AT %X28.1 : BOOL;
	        Signals_28_2 AT %X28.2 : BOOL;
	        Signals_28_3 AT %X28.3 : BOOL;
	        Signals_28_4 AT %X28.4 : BOOL;
	        Signals_28_5 AT %X28.5 : BOOL;
	        Signals_28_6 AT %X28.6 : BOOL;
	        Signals_28_7 AT %X28.7 : BOOL;
	        Signals_29_0 AT %X29.0 : BOOL;
	        Signals_29_1 AT %X29.1 : BOOL;
	        Signals_29_2 AT %X29.2 : BOOL;
	        Signals_29_3 AT %X29.3 : BOOL;
	        Signals_29_4 AT %X29.4 : BOOL;
	        Signals_29_5 AT %X29.5 : BOOL;
	        Signals_29_6 AT %X29.6 : BOOL;
	        Signals_29_7 AT %X29.7 : BOOL;
	        Signals_30_0 AT %X30.0 : BOOL;
	        Signals_30_1 AT %X30.1 : BOOL;
	        Signals_30_2 AT %X30.2 : BOOL;
	        Signals_30_3 AT %X30.3 : BOOL;
	        Signals_30_4 AT %X30.4 : BOOL;
	        Signals_30_5 AT %X30.5 : BOOL;
	        Signals_30_6 AT %X30.6 : BOOL;
	        Signals_30_7 AT %X30.7 : BOOL;
	        Signals_31_0 AT %X31.0 : BOOL;
	        Signals_31_1 AT %X31.1 : BOOL;
	        Signals_31_2 AT %X31.2 : BOOL;
	        Signals_31_3 AT %X31.3 : BOOL;
	        Signals_31_4 AT %X31.4 : BOOL;
	        Signals_31_5 AT %X31.5 : BOOL;
	        Signals_31_6 AT %X31.6 : BOOL;
	        Signals_31_7 AT %X31.7 : BOOL;
	        Signals_32_0 AT %X32.0 : BOOL;
	        Signals_32_1 AT %X32.1 : BOOL;
	        Signals_32_2 AT %X32.2 : BOOL;
	        Signals_32_3 AT %X32.3 : BOOL;
	        Signals_32_4 AT %X32.4 : BOOL;
	        Signals_32_5 AT %X32.5 : BOOL;
	        Signals_32_6 AT %X32.6 : BOOL;
	        Signals_32_7 AT %X32.7 : BOOL;
	        Signals_33_0 AT %X33.0 : BOOL;
	        Signals_33_1 AT %X33.1 : BOOL;
	        Signals_33_2 AT %X33.2 : BOOL;
	        Signals_33_3 AT %X33.3 : BOOL;
	        Signals_33_4 AT %X33.4 : BOOL;
	        Signals_33_5 AT %X33.5 : BOOL;
	        Signals_33_6 AT %X33.6 : BOOL;
	        Signals_33_7 AT %X33.7 : BOOL;
	        Signals_34_0 AT %X34.0 : BOOL;
	        Signals_34_1 AT %X34.1 : BOOL;
	        Signals_34_2 AT %X34.2 : BOOL;
	        Signals_34_3 AT %X34.3 : BOOL;
	        Signals_34_4 AT %X34.4 : BOOL;
	        Signals_34_5 AT %X34.5 : BOOL;
	        Signals_34_6 AT %X34.6 : BOOL;
	        Signals_34_7 AT %X34.7 : BOOL;
	        Signals_35_0 AT %X35.0 : BOOL;
	        Signals_35_1 AT %X35.1 : BOOL;
	        Signals_35_2 AT %X35.2 : BOOL;
	        Signals_35_3 AT %X35.3 : BOOL;
	        Signals_35_4 AT %X35.4 : BOOL;
	        Signals_35_5 AT %X35.5 : BOOL;
	        Signals_35_6 AT %X35.6 : BOOL;
	        Signals_35_7 AT %X35.7 : BOOL;
	        Signals_36_0 AT %X36.0 : BOOL;
	        Signals_36_1 AT %X36.1 : BOOL;
	        Signals_36_2 AT %X36.2 : BOOL;
	        Signals_36_3 AT %X36.3 : BOOL;
	        Signals_36_4 AT %X36.4 : BOOL;
	        Signals_36_5 AT %X36.5 : BOOL;
	        Signals_36_6 AT %X36.6 : BOOL;
	        Signals_36_7 AT %X36.7 : BOOL;
	        Signals_37_0 AT %X37.0 : BOOL;
	        Signals_37_1 AT %X37.1 : BOOL;
	        Signals_37_2 AT %X37.2 : BOOL;
	        Signals_37_3 AT %X37.3 : BOOL;
	        Signals_37_4 AT %X37.4 : BOOL;
	        Signals_37_5 AT %X37.5 : BOOL;
	        Signals_37_6 AT %X37.6 : BOOL;
	        Signals_37_7 AT %X37.7 : BOOL;
	        Signals_38_0 AT %X38.0 : BOOL;
	        Signals_38_1 AT %X38.1 : BOOL;
	        Signals_38_2 AT %X38.2 : BOOL;
	        Signals_38_3 AT %X38.3 : BOOL;
	        Signals_38_4 AT %X38.4 : BOOL;
	        Signals_38_5 AT %X38.5 : BOOL;
	        Signals_38_6 AT %X38.6 : BOOL;
	        Signals_38_7 AT %X38.7 : BOOL;
	        Signals_39_0 AT %X39.0 : BOOL;
	        Signals_39_1 AT %X39.1 : BOOL;
	        Signals_39_2 AT %X39.2 : BOOL;
	        Signals_39_3 AT %X39.3 : BOOL;
	        Signals_39_4 AT %X39.4 : BOOL;
	        Signals_39_5 AT %X39.5 : BOOL;
	        Signals_39_6 AT %X39.6 : BOOL;
	        Signals_39_7 AT %X39.7 : BOOL;
	        Signals_40_0 AT %X40.0 : BOOL;
	        Signals_40_1 AT %X40.1 : BOOL;
	        Signals_40_2 AT %X40.2 : BOOL;
	        Signals_40_3 AT %X40.3 : BOOL;
	        Signals_40_4 AT %X40.4 : BOOL;
	        Signals_40_5 AT %X40.5 : BOOL;
	        Signals_40_6 AT %X40.6 : BOOL;
	        Signals_40_7 AT %X40.7 : BOOL;
	        Signals_41_0 AT %X41.0 : BOOL;
	        Signals_41_1 AT %X41.1 : BOOL;
	        Signals_41_2 AT %X41.2 : BOOL;
	        Signals_41_3 AT %X41.3 : BOOL;
	        Signals_41_4 AT %X41.4 : BOOL;
	        Signals_41_5 AT %X41.5 : BOOL;
	        Signals_41_6 AT %X41.6 : BOOL;
	        Signals_41_7 AT %X41.7 : BOOL;
	        Signals_42_0 AT %X42.0 : BOOL;
	        Signals_42_1 AT %X42.1 : BOOL;
	        Signals_42_2 AT %X42.2 : BOOL;
	        Signals_42_3 AT %X42.3 : BOOL;
	        Signals_42_4 AT %X42.4 : BOOL;
	        Signals_42_5 AT %X42.5 : BOOL;
	        Signals_42_6 AT %X42.6 : BOOL;
	        Signals_42_7 AT %X42.7 : BOOL;
	        Signals_43_0 AT %X43.0 : BOOL;
	        Signals_43_1 AT %X43.1 : BOOL;
	        Signals_43_2 AT %X43.2 : BOOL;
	        Signals_43_3 AT %X43.3 : BOOL;
	        Signals_43_4 AT %X43.4 : BOOL;
	        Signals_43_5 AT %X43.5 : BOOL;
	        Signals_43_6 AT %X43.6 : BOOL;
	        Signals_43_7 AT %X43.7 : BOOL;
	        Signals_44_0 AT %X44.0 : BOOL;
	        Signals_44_1 AT %X44.1 : BOOL;
	        Signals_44_2 AT %X44.2 : BOOL;
	        Signals_44_3 AT %X44.3 : BOOL;
	        Signals_44_4 AT %X44.4 : BOOL;
	        Signals_44_5 AT %X44.5 : BOOL;
	        Signals_44_6 AT %X44.6 : BOOL;
	        Signals_44_7 AT %X44.7 : BOOL;
	        Signals_45_0 AT %X45.0 : BOOL;
	        Signals_45_1 AT %X45.1 : BOOL;
	        Signals_45_2 AT %X45.2 : BOOL;
	        Signals_45_3 AT %X45.3 : BOOL;
	        Signals_45_4 AT %X45.4 : BOOL;
	        Signals_45_5 AT %X45.5 : BOOL;
	        Signals_45_6 AT %X45.6 : BOOL;
	        Signals_45_7 AT %X45.7 : BOOL;
	        Signals_46_0 AT %X46.0 : BOOL;
	        Signals_46_1 AT %X46.1 : BOOL;
	        Signals_46_2 AT %X46.2 : BOOL;
	        Signals_46_3 AT %X46.3 : BOOL;
	        Signals_46_4 AT %X46.4 : BOOL;
	        Signals_46_5 AT %X46.5 : BOOL;
	        Signals_46_6 AT %X46.6 : BOOL;
	        Signals_46_7 AT %X46.7 : BOOL;
	        Signals_47_0 AT %X47.0 : BOOL;
	        Signals_47_1 AT %X47.1 : BOOL;
	        Signals_47_2 AT %X47.2 : BOOL;
	        Signals_47_3 AT %X47.3 : BOOL;
	        Signals_47_4 AT %X47.4 : BOOL;
	        Signals_47_5 AT %X47.5 : BOOL;
	        Signals_47_6 AT %X47.6 : BOOL;
	        Signals_47_7 AT %X47.7 : BOOL;
	        Signals_48_0 AT %X48.0 : BOOL;
	        Signals_48_1 AT %X48.1 : BOOL;
	        Signals_48_2 AT %X48.2 : BOOL;
	        Signals_48_3 AT %X48.3 : BOOL;
	        Signals_48_4 AT %X48.4 : BOOL;
	        Signals_48_5 AT %X48.5 : BOOL;
	        Signals_48_6 AT %X48.6 : BOOL;
	        Signals_48_7 AT %X48.7 : BOOL;
	        Signals_49_0 AT %X49.0 : BOOL;
	        Signals_49_1 AT %X49.1 : BOOL;
	        Signals_49_2 AT %X49.2 : BOOL;
	        Signals_49_3 AT %X49.3 : BOOL;
	        Signals_49_4 AT %X49.4 : BOOL;
	        Signals_49_5 AT %X49.5 : BOOL;
	        Signals_49_6 AT %X49.6 : BOOL;
	        Signals_49_7 AT %X49.7 : BOOL;
	        Signals_50_0 AT %X50.0 : BOOL;
	        Signals_50_1 AT %X50.1 : BOOL;
	        Signals_50_2 AT %X50.2 : BOOL;
	        Signals_50_3 AT %X50.3 : BOOL;
	        Signals_50_4 AT %X50.4 : BOOL;
	        Signals_50_5 AT %X50.5 : BOOL;
	        Signals_50_6 AT %X50.6 : BOOL;
	        Signals_50_7 AT %X50.7 : BOOL;
	        Signals_51_0 AT %X51.0 : BOOL;
	        Signals_51_1 AT %X51.1 : BOOL;
	        Signals_51_2 AT %X51.2 : BOOL;
	        Signals_51_3 AT %X51.3 : BOOL;
	        Signals_51_4 AT %X51.4 : BOOL;
	        Signals_51_5 AT %X51.5 : BOOL;
	        Signals_51_6 AT %X51.6 : BOOL;
	        Signals_51_7 AT %X51.7 : BOOL;
	        Signals_52_0 AT %X52.0 : BOOL;
	        Signals_52_1 AT %X52.1 : BOOL;
	        Signals_52_2 AT %X52.2 : BOOL;
	        Signals_52_3 AT %X52.3 : BOOL;
	        Signals_52_4 AT %X52.4 : BOOL;
	        Signals_52_5 AT %X52.5 : BOOL;
	        Signals_52_6 AT %X52.6 : BOOL;
	        Signals_52_7 AT %X52.7 : BOOL;
	        Signals_53_0 AT %X53.0 : BOOL;
	        Signals_53_1 AT %X53.1 : BOOL;
	        Signals_53_2 AT %X53.2 : BOOL;
	        Signals_53_3 AT %X53.3 : BOOL;
	        Signals_53_4 AT %X53.4 : BOOL;
	        Signals_53_5 AT %X53.5 : BOOL;
	        Signals_53_6 AT %X53.6 : BOOL;
	        Signals_53_7 AT %X53.7 : BOOL;
	        Signals_54_0 AT %X54.0 : BOOL;
	        Signals_54_1 AT %X54.1 : BOOL;
	        Signals_54_2 AT %X54.2 : BOOL;
	        Signals_54_3 AT %X54.3 : BOOL;
	        Signals_54_4 AT %X54.4 : BOOL;
	        Signals_54_5 AT %X54.5 : BOOL;
	        Signals_54_6 AT %X54.6 : BOOL;
	        Signals_54_7 AT %X54.7 : BOOL;
	        Signals_55_0 AT %X55.0 : BOOL;
	        Signals_55_1 AT %X55.1 : BOOL;
	        Signals_55_2 AT %X55.2 : BOOL;
	        Signals_55_3 AT %X55.3 : BOOL;
	        Signals_55_4 AT %X55.4 : BOOL;
	        Signals_55_5 AT %X55.5 : BOOL;
	        Signals_55_6 AT %X55.6 : BOOL;
	        Signals_55_7 AT %X55.7 : BOOL;
	        Signals_56_0 AT %X56.0 : BOOL;
	        Signals_56_1 AT %X56.1 : BOOL;
	        Signals_56_2 AT %X56.2 : BOOL;
	        Signals_56_3 AT %X56.3 : BOOL;
	        Signals_56_4 AT %X56.4 : BOOL;
	        Signals_56_5 AT %X56.5 : BOOL;
	        Signals_56_6 AT %X56.6 : BOOL;
	        Signals_56_7 AT %X56.7 : BOOL;
	        Signals_57_0 AT %X57.0 : BOOL;
	        Signals_57_1 AT %X57.1 : BOOL;
	        Signals_57_2 AT %X57.2 : BOOL;
	        Signals_57_3 AT %X57.3 : BOOL;
	        Signals_57_4 AT %X57.4 : BOOL;
	        Signals_57_5 AT %X57.5 : BOOL;
	        Signals_57_6 AT %X57.6 : BOOL;
	        Signals_57_7 AT %X57.7 : BOOL;
	        Signals_58_0 AT %X58.0 : BOOL;
	        Signals_58_1 AT %X58.1 : BOOL;
	        Signals_58_2 AT %X58.2 : BOOL;
	        Signals_58_3 AT %X58.3 : BOOL;
	        Signals_58_4 AT %X58.4 : BOOL;
	        Signals_58_5 AT %X58.5 : BOOL;
	        Signals_58_6 AT %X58.6 : BOOL;
	        Signals_58_7 AT %X58.7 : BOOL;
	        Signals_59_0 AT %X59.0 : BOOL;
	        Signals_59_1 AT %X59.1 : BOOL;
	        Signals_59_2 AT %X59.2 : BOOL;
	        Signals_59_3 AT %X59.3 : BOOL;
	        Signals_59_4 AT %X59.4 : BOOL;
	        Signals_59_5 AT %X59.5 : BOOL;
	        Signals_59_6 AT %X59.6 : BOOL;
	        Signals_59_7 AT %X59.7 : BOOL;
	        Signals_60_0 AT %X60.0 : BOOL;
	        Signals_60_1 AT %X60.1 : BOOL;
	        Signals_60_2 AT %X60.2 : BOOL;
	        Signals_60_3 AT %X60.3 : BOOL;
	        Signals_60_4 AT %X60.4 : BOOL;
	        Signals_60_5 AT %X60.5 : BOOL;
	        Signals_60_6 AT %X60.6 : BOOL;
	        Signals_60_7 AT %X60.7 : BOOL;
	        Signals_61_0 AT %X61.0 : BOOL;
	        Signals_61_1 AT %X61.1 : BOOL;
	        Signals_61_2 AT %X61.2 : BOOL;
	        Signals_61_3 AT %X61.3 : BOOL;
	        Signals_61_4 AT %X61.4 : BOOL;
	        Signals_61_5 AT %X61.5 : BOOL;
	        Signals_61_6 AT %X61.6 : BOOL;
	        Signals_61_7 AT %X61.7 : BOOL;
	        Signals_62_0 AT %X62.0 : BOOL;
	        Signals_62_1 AT %X62.1 : BOOL;
	        Signals_62_2 AT %X62.2 : BOOL;
	        Signals_62_3 AT %X62.3 : BOOL;
	        Signals_62_4 AT %X62.4 : BOOL;
	        Signals_62_5 AT %X62.5 : BOOL;
	        Signals_62_6 AT %X62.6 : BOOL;
	        Signals_62_7 AT %X62.7 : BOOL;
	        Signals_63_0 AT %X63.0 : BOOL;
	        Signals_63_1 AT %X63.1 : BOOL;
	        Signals_63_2 AT %X63.2 : BOOL;
	        Signals_63_3 AT %X63.3 : BOOL;
	        Signals_63_4 AT %X63.4 : BOOL;
	        Signals_63_5 AT %X63.5 : BOOL;
	        Signals_63_6 AT %X63.6 : BOOL;
	        Signals_63_7 AT %X63.7 : BOOL;
	    END_STRUCT;
	END_TYPE

	TYPE
        {S7.extern=ReadWrite}
        {#ix-attr:[Container(Layout.Wrap)]}
	    kuka_rb1_DIO512_Output_Layout : STRUCT
	        Signals_64_0 AT %X0.0 : BOOL;
	        Signals_64_1 AT %X0.1 : BOOL;
	        Signals_64_2 AT %X0.2 : BOOL;
	        Signals_64_3 AT %X0.3 : BOOL;
	        Signals_64_4 AT %X0.4 : BOOL;
	        Signals_64_5 AT %X0.5 : BOOL;
	        Signals_64_6 AT %X0.6 : BOOL;
	        Signals_64_7 AT %X0.7 : BOOL;
	        Signals_65_0 AT %X1.0 : BOOL;
	        Signals_65_1 AT %X1.1 : BOOL;
	        Signals_65_2 AT %X1.2 : BOOL;
	        Signals_65_3 AT %X1.3 : BOOL;
	        Signals_65_4 AT %X1.4 : BOOL;
	        Signals_65_5 AT %X1.5 : BOOL;
	        Signals_65_6 AT %X1.6 : BOOL;
	        Signals_65_7 AT %X1.7 : BOOL;
	        Signals_66_0 AT %X2.0 : BOOL;
	        Signals_66_1 AT %X2.1 : BOOL;
	        Signals_66_2 AT %X2.2 : BOOL;
	        Signals_66_3 AT %X2.3 : BOOL;
	        Signals_66_4 AT %X2.4 : BOOL;
	        Signals_66_5 AT %X2.5 : BOOL;
	        Signals_66_6 AT %X2.6 : BOOL;
	        Signals_66_7 AT %X2.7 : BOOL;
	        Signals_67_0 AT %X3.0 : BOOL;
	        Signals_67_1 AT %X3.1 : BOOL;
	        Signals_67_2 AT %X3.2 : BOOL;
	        Signals_67_3 AT %X3.3 : BOOL;
	        Signals_67_4 AT %X3.4 : BOOL;
	        Signals_67_5 AT %X3.5 : BOOL;
	        Signals_67_6 AT %X3.6 : BOOL;
	        Signals_67_7 AT %X3.7 : BOOL;
	        Signals_68_0 AT %X4.0 : BOOL;
	        Signals_68_1 AT %X4.1 : BOOL;
	        Signals_68_2 AT %X4.2 : BOOL;
	        Signals_68_3 AT %X4.3 : BOOL;
	        Signals_68_4 AT %X4.4 : BOOL;
	        Signals_68_5 AT %X4.5 : BOOL;
	        Signals_68_6 AT %X4.6 : BOOL;
	        Signals_68_7 AT %X4.7 : BOOL;
	        Signals_69_0 AT %X5.0 : BOOL;
	        Signals_69_1 AT %X5.1 : BOOL;
	        Signals_69_2 AT %X5.2 : BOOL;
	        Signals_69_3 AT %X5.3 : BOOL;
	        Signals_69_4 AT %X5.4 : BOOL;
	        Signals_69_5 AT %X5.5 : BOOL;
	        Signals_69_6 AT %X5.6 : BOOL;
	        Signals_69_7 AT %X5.7 : BOOL;
	        Signals_70_0 AT %X6.0 : BOOL;
	        Signals_70_1 AT %X6.1 : BOOL;
	        Signals_70_2 AT %X6.2 : BOOL;
	        Signals_70_3 AT %X6.3 : BOOL;
	        Signals_70_4 AT %X6.4 : BOOL;
	        Signals_70_5 AT %X6.5 : BOOL;
	        Signals_70_6 AT %X6.6 : BOOL;
	        Signals_70_7 AT %X6.7 : BOOL;
	        Signals_71_0 AT %X7.0 : BOOL;
	        Signals_71_1 AT %X7.1 : BOOL;
	        Signals_71_2 AT %X7.2 : BOOL;
	        Signals_71_3 AT %X7.3 : BOOL;
	        Signals_71_4 AT %X7.4 : BOOL;
	        Signals_71_5 AT %X7.5 : BOOL;
	        Signals_71_6 AT %X7.6 : BOOL;
	        Signals_71_7 AT %X7.7 : BOOL;
	        Signals_72_0 AT %X8.0 : BOOL;
	        Signals_72_1 AT %X8.1 : BOOL;
	        Signals_72_2 AT %X8.2 : BOOL;
	        Signals_72_3 AT %X8.3 : BOOL;
	        Signals_72_4 AT %X8.4 : BOOL;
	        Signals_72_5 AT %X8.5 : BOOL;
	        Signals_72_6 AT %X8.6 : BOOL;
	        Signals_72_7 AT %X8.7 : BOOL;
	        Signals_73_0 AT %X9.0 : BOOL;
	        Signals_73_1 AT %X9.1 : BOOL;
	        Signals_73_2 AT %X9.2 : BOOL;
	        Signals_73_3 AT %X9.3 : BOOL;
	        Signals_73_4 AT %X9.4 : BOOL;
	        Signals_73_5 AT %X9.5 : BOOL;
	        Signals_73_6 AT %X9.6 : BOOL;
	        Signals_73_7 AT %X9.7 : BOOL;
	        Signals_74_0 AT %X10.0 : BOOL;
	        Signals_74_1 AT %X10.1 : BOOL;
	        Signals_74_2 AT %X10.2 : BOOL;
	        Signals_74_3 AT %X10.3 : BOOL;
	        Signals_74_4 AT %X10.4 : BOOL;
	        Signals_74_5 AT %X10.5 : BOOL;
	        Signals_74_6 AT %X10.6 : BOOL;
	        Signals_74_7 AT %X10.7 : BOOL;
	        Signals_75_0 AT %X11.0 : BOOL;
	        Signals_75_1 AT %X11.1 : BOOL;
	        Signals_75_2 AT %X11.2 : BOOL;
	        Signals_75_3 AT %X11.3 : BOOL;
	        Signals_75_4 AT %X11.4 : BOOL;
	        Signals_75_5 AT %X11.5 : BOOL;
	        Signals_75_6 AT %X11.6 : BOOL;
	        Signals_75_7 AT %X11.7 : BOOL;
	        Signals_76_0 AT %X12.0 : BOOL;
	        Signals_76_1 AT %X12.1 : BOOL;
	        Signals_76_2 AT %X12.2 : BOOL;
	        Signals_76_3 AT %X12.3 : BOOL;
	        Signals_76_4 AT %X12.4 : BOOL;
	        Signals_76_5 AT %X12.5 : BOOL;
	        Signals_76_6 AT %X12.6 : BOOL;
	        Signals_76_7 AT %X12.7 : BOOL;
	        Signals_77_0 AT %X13.0 : BOOL;
	        Signals_77_1 AT %X13.1 : BOOL;
	        Signals_77_2 AT %X13.2 : BOOL;
	        Signals_77_3 AT %X13.3 : BOOL;
	        Signals_77_4 AT %X13.4 : BOOL;
	        Signals_77_5 AT %X13.5 : BOOL;
	        Signals_77_6 AT %X13.6 : BOOL;
	        Signals_77_7 AT %X13.7 : BOOL;
	        Signals_78_0 AT %X14.0 : BOOL;
	        Signals_78_1 AT %X14.1 : BOOL;
	        Signals_78_2 AT %X14.2 : BOOL;
	        Signals_78_3 AT %X14.3 : BOOL;
	        Signals_78_4 AT %X14.4 : BOOL;
	        Signals_78_5 AT %X14.5 : BOOL;
	        Signals_78_6 AT %X14.6 : BOOL;
	        Signals_78_7 AT %X14.7 : BOOL;
	        Signals_79_0 AT %X15.0 : BOOL;
	        Signals_79_1 AT %X15.1 : BOOL;
	        Signals_79_2 AT %X15.2 : BOOL;
	        Signals_79_3 AT %X15.3 : BOOL;
	        Signals_79_4 AT %X15.4 : BOOL;
	        Signals_79_5 AT %X15.5 : BOOL;
	        Signals_79_6 AT %X15.6 : BOOL;
	        Signals_79_7 AT %X15.7 : BOOL;
	        Signals_80_0 AT %X16.0 : BOOL;
	        Signals_80_1 AT %X16.1 : BOOL;
	        Signals_80_2 AT %X16.2 : BOOL;
	        Signals_80_3 AT %X16.3 : BOOL;
	        Signals_80_4 AT %X16.4 : BOOL;
	        Signals_80_5 AT %X16.5 : BOOL;
	        Signals_80_6 AT %X16.6 : BOOL;
	        Signals_80_7 AT %X16.7 : BOOL;
	        Signals_81_0 AT %X17.0 : BOOL;
	        Signals_81_1 AT %X17.1 : BOOL;
	        Signals_81_2 AT %X17.2 : BOOL;
	        Signals_81_3 AT %X17.3 : BOOL;
	        Signals_81_4 AT %X17.4 : BOOL;
	        Signals_81_5 AT %X17.5 : BOOL;
	        Signals_81_6 AT %X17.6 : BOOL;
	        Signals_81_7 AT %X17.7 : BOOL;
	        Signals_82_0 AT %X18.0 : BOOL;
	        Signals_82_1 AT %X18.1 : BOOL;
	        Signals_82_2 AT %X18.2 : BOOL;
	        Signals_82_3 AT %X18.3 : BOOL;
	        Signals_82_4 AT %X18.4 : BOOL;
	        Signals_82_5 AT %X18.5 : BOOL;
	        Signals_82_6 AT %X18.6 : BOOL;
	        Signals_82_7 AT %X18.7 : BOOL;
	        Signals_83_0 AT %X19.0 : BOOL;
	        Signals_83_1 AT %X19.1 : BOOL;
	        Signals_83_2 AT %X19.2 : BOOL;
	        Signals_83_3 AT %X19.3 : BOOL;
	        Signals_83_4 AT %X19.4 : BOOL;
	        Signals_83_5 AT %X19.5 : BOOL;
	        Signals_83_6 AT %X19.6 : BOOL;
	        Signals_83_7 AT %X19.7 : BOOL;
	        Signals_84_0 AT %X20.0 : BOOL;
	        Signals_84_1 AT %X20.1 : BOOL;
	        Signals_84_2 AT %X20.2 : BOOL;
	        Signals_84_3 AT %X20.3 : BOOL;
	        Signals_84_4 AT %X20.4 : BOOL;
	        Signals_84_5 AT %X20.5 : BOOL;
	        Signals_84_6 AT %X20.6 : BOOL;
	        Signals_84_7 AT %X20.7 : BOOL;
	        Signals_85_0 AT %X21.0 : BOOL;
	        Signals_85_1 AT %X21.1 : BOOL;
	        Signals_85_2 AT %X21.2 : BOOL;
	        Signals_85_3 AT %X21.3 : BOOL;
	        Signals_85_4 AT %X21.4 : BOOL;
	        Signals_85_5 AT %X21.5 : BOOL;
	        Signals_85_6 AT %X21.6 : BOOL;
	        Signals_85_7 AT %X21.7 : BOOL;
	        Signals_86_0 AT %X22.0 : BOOL;
	        Signals_86_1 AT %X22.1 : BOOL;
	        Signals_86_2 AT %X22.2 : BOOL;
	        Signals_86_3 AT %X22.3 : BOOL;
	        Signals_86_4 AT %X22.4 : BOOL;
	        Signals_86_5 AT %X22.5 : BOOL;
	        Signals_86_6 AT %X22.6 : BOOL;
	        Signals_86_7 AT %X22.7 : BOOL;
	        Signals_87_0 AT %X23.0 : BOOL;
	        Signals_87_1 AT %X23.1 : BOOL;
	        Signals_87_2 AT %X23.2 : BOOL;
	        Signals_87_3 AT %X23.3 : BOOL;
	        Signals_87_4 AT %X23.4 : BOOL;
	        Signals_87_5 AT %X23.5 : BOOL;
	        Signals_87_6 AT %X23.6 : BOOL;
	        Signals_87_7 AT %X23.7 : BOOL;
	        Signals_88_0 AT %X24.0 : BOOL;
	        Signals_88_1 AT %X24.1 : BOOL;
	        Signals_88_2 AT %X24.2 : BOOL;
	        Signals_88_3 AT %X24.3 : BOOL;
	        Signals_88_4 AT %X24.4 : BOOL;
	        Signals_88_5 AT %X24.5 : BOOL;
	        Signals_88_6 AT %X24.6 : BOOL;
	        Signals_88_7 AT %X24.7 : BOOL;
	        Signals_89_0 AT %X25.0 : BOOL;
	        Signals_89_1 AT %X25.1 : BOOL;
	        Signals_89_2 AT %X25.2 : BOOL;
	        Signals_89_3 AT %X25.3 : BOOL;
	        Signals_89_4 AT %X25.4 : BOOL;
	        Signals_89_5 AT %X25.5 : BOOL;
	        Signals_89_6 AT %X25.6 : BOOL;
	        Signals_89_7 AT %X25.7 : BOOL;
	        Signals_90_0 AT %X26.0 : BOOL;
	        Signals_90_1 AT %X26.1 : BOOL;
	        Signals_90_2 AT %X26.2 : BOOL;
	        Signals_90_3 AT %X26.3 : BOOL;
	        Signals_90_4 AT %X26.4 : BOOL;
	        Signals_90_5 AT %X26.5 : BOOL;
	        Signals_90_6 AT %X26.6 : BOOL;
	        Signals_90_7 AT %X26.7 : BOOL;
	        Signals_91_0 AT %X27.0 : BOOL;
	        Signals_91_1 AT %X27.1 : BOOL;
	        Signals_91_2 AT %X27.2 : BOOL;
	        Signals_91_3 AT %X27.3 : BOOL;
	        Signals_91_4 AT %X27.4 : BOOL;
	        Signals_91_5 AT %X27.5 : BOOL;
	        Signals_91_6 AT %X27.6 : BOOL;
	        Signals_91_7 AT %X27.7 : BOOL;
	        Signals_92_0 AT %X28.0 : BOOL;
	        Signals_92_1 AT %X28.1 : BOOL;
	        Signals_92_2 AT %X28.2 : BOOL;
	        Signals_92_3 AT %X28.3 : BOOL;
	        Signals_92_4 AT %X28.4 : BOOL;
	        Signals_92_5 AT %X28.5 : BOOL;
	        Signals_92_6 AT %X28.6 : BOOL;
	        Signals_92_7 AT %X28.7 : BOOL;
	        Signals_93_0 AT %X29.0 : BOOL;
	        Signals_93_1 AT %X29.1 : BOOL;
	        Signals_93_2 AT %X29.2 : BOOL;
	        Signals_93_3 AT %X29.3 : BOOL;
	        Signals_93_4 AT %X29.4 : BOOL;
	        Signals_93_5 AT %X29.5 : BOOL;
	        Signals_93_6 AT %X29.6 : BOOL;
	        Signals_93_7 AT %X29.7 : BOOL;
	        Signals_94_0 AT %X30.0 : BOOL;
	        Signals_94_1 AT %X30.1 : BOOL;
	        Signals_94_2 AT %X30.2 : BOOL;
	        Signals_94_3 AT %X30.3 : BOOL;
	        Signals_94_4 AT %X30.4 : BOOL;
	        Signals_94_5 AT %X30.5 : BOOL;
	        Signals_94_6 AT %X30.6 : BOOL;
	        Signals_94_7 AT %X30.7 : BOOL;
	        Signals_95_0 AT %X31.0 : BOOL;
	        Signals_95_1 AT %X31.1 : BOOL;
	        Signals_95_2 AT %X31.2 : BOOL;
	        Signals_95_3 AT %X31.3 : BOOL;
	        Signals_95_4 AT %X31.4 : BOOL;
	        Signals_95_5 AT %X31.5 : BOOL;
	        Signals_95_6 AT %X31.6 : BOOL;
	        Signals_95_7 AT %X31.7 : BOOL;
	        Signals_96_0 AT %X32.0 : BOOL;
	        Signals_96_1 AT %X32.1 : BOOL;
	        Signals_96_2 AT %X32.2 : BOOL;
	        Signals_96_3 AT %X32.3 : BOOL;
	        Signals_96_4 AT %X32.4 : BOOL;
	        Signals_96_5 AT %X32.5 : BOOL;
	        Signals_96_6 AT %X32.6 : BOOL;
	        Signals_96_7 AT %X32.7 : BOOL;
	        Signals_97_0 AT %X33.0 : BOOL;
	        Signals_97_1 AT %X33.1 : BOOL;
	        Signals_97_2 AT %X33.2 : BOOL;
	        Signals_97_3 AT %X33.3 : BOOL;
	        Signals_97_4 AT %X33.4 : BOOL;
	        Signals_97_5 AT %X33.5 : BOOL;
	        Signals_97_6 AT %X33.6 : BOOL;
	        Signals_97_7 AT %X33.7 : BOOL;
	        Signals_98_0 AT %X34.0 : BOOL;
	        Signals_98_1 AT %X34.1 : BOOL;
	        Signals_98_2 AT %X34.2 : BOOL;
	        Signals_98_3 AT %X34.3 : BOOL;
	        Signals_98_4 AT %X34.4 : BOOL;
	        Signals_98_5 AT %X34.5 : BOOL;
	        Signals_98_6 AT %X34.6 : BOOL;
	        Signals_98_7 AT %X34.7 : BOOL;
	        Signals_99_0 AT %X35.0 : BOOL;
	        Signals_99_1 AT %X35.1 : BOOL;
	        Signals_99_2 AT %X35.2 : BOOL;
	        Signals_99_3 AT %X35.3 : BOOL;
	        Signals_99_4 AT %X35.4 : BOOL;
	        Signals_99_5 AT %X35.5 : BOOL;
	        Signals_99_6 AT %X35.6 : BOOL;
	        Signals_99_7 AT %X35.7 : BOOL;
	        Signals_100_0 AT %X36.0 : BOOL;
	        Signals_100_1 AT %X36.1 : BOOL;
	        Signals_100_2 AT %X36.2 : BOOL;
	        Signals_100_3 AT %X36.3 : BOOL;
	        Signals_100_4 AT %X36.4 : BOOL;
	        Signals_100_5 AT %X36.5 : BOOL;
	        Signals_100_6 AT %X36.6 : BOOL;
	        Signals_100_7 AT %X36.7 : BOOL;
	        Signals_101_0 AT %X37.0 : BOOL;
	        Signals_101_1 AT %X37.1 : BOOL;
	        Signals_101_2 AT %X37.2 : BOOL;
	        Signals_101_3 AT %X37.3 : BOOL;
	        Signals_101_4 AT %X37.4 : BOOL;
	        Signals_101_5 AT %X37.5 : BOOL;
	        Signals_101_6 AT %X37.6 : BOOL;
	        Signals_101_7 AT %X37.7 : BOOL;
	        Signals_102_0 AT %X38.0 : BOOL;
	        Signals_102_1 AT %X38.1 : BOOL;
	        Signals_102_2 AT %X38.2 : BOOL;
	        Signals_102_3 AT %X38.3 : BOOL;
	        Signals_102_4 AT %X38.4 : BOOL;
	        Signals_102_5 AT %X38.5 : BOOL;
	        Signals_102_6 AT %X38.6 : BOOL;
	        Signals_102_7 AT %X38.7 : BOOL;
	        Signals_103_0 AT %X39.0 : BOOL;
	        Signals_103_1 AT %X39.1 : BOOL;
	        Signals_103_2 AT %X39.2 : BOOL;
	        Signals_103_3 AT %X39.3 : BOOL;
	        Signals_103_4 AT %X39.4 : BOOL;
	        Signals_103_5 AT %X39.5 : BOOL;
	        Signals_103_6 AT %X39.6 : BOOL;
	        Signals_103_7 AT %X39.7 : BOOL;
	        Signals_104_0 AT %X40.0 : BOOL;
	        Signals_104_1 AT %X40.1 : BOOL;
	        Signals_104_2 AT %X40.2 : BOOL;
	        Signals_104_3 AT %X40.3 : BOOL;
	        Signals_104_4 AT %X40.4 : BOOL;
	        Signals_104_5 AT %X40.5 : BOOL;
	        Signals_104_6 AT %X40.6 : BOOL;
	        Signals_104_7 AT %X40.7 : BOOL;
	        Signals_105_0 AT %X41.0 : BOOL;
	        Signals_105_1 AT %X41.1 : BOOL;
	        Signals_105_2 AT %X41.2 : BOOL;
	        Signals_105_3 AT %X41.3 : BOOL;
	        Signals_105_4 AT %X41.4 : BOOL;
	        Signals_105_5 AT %X41.5 : BOOL;
	        Signals_105_6 AT %X41.6 : BOOL;
	        Signals_105_7 AT %X41.7 : BOOL;
	        Signals_106_0 AT %X42.0 : BOOL;
	        Signals_106_1 AT %X42.1 : BOOL;
	        Signals_106_2 AT %X42.2 : BOOL;
	        Signals_106_3 AT %X42.3 : BOOL;
	        Signals_106_4 AT %X42.4 : BOOL;
	        Signals_106_5 AT %X42.5 : BOOL;
	        Signals_106_6 AT %X42.6 : BOOL;
	        Signals_106_7 AT %X42.7 : BOOL;
	        Signals_107_0 AT %X43.0 : BOOL;
	        Signals_107_1 AT %X43.1 : BOOL;
	        Signals_107_2 AT %X43.2 : BOOL;
	        Signals_107_3 AT %X43.3 : BOOL;
	        Signals_107_4 AT %X43.4 : BOOL;
	        Signals_107_5 AT %X43.5 : BOOL;
	        Signals_107_6 AT %X43.6 : BOOL;
	        Signals_107_7 AT %X43.7 : BOOL;
	        Signals_108_0 AT %X44.0 : BOOL;
	        Signals_108_1 AT %X44.1 : BOOL;
	        Signals_108_2 AT %X44.2 : BOOL;
	        Signals_108_3 AT %X44.3 : BOOL;
	        Signals_108_4 AT %X44.4 : BOOL;
	        Signals_108_5 AT %X44.5 : BOOL;
	        Signals_108_6 AT %X44.6 : BOOL;
	        Signals_108_7 AT %X44.7 : BOOL;
	        Signals_109_0 AT %X45.0 : BOOL;
	        Signals_109_1 AT %X45.1 : BOOL;
	        Signals_109_2 AT %X45.2 : BOOL;
	        Signals_109_3 AT %X45.3 : BOOL;
	        Signals_109_4 AT %X45.4 : BOOL;
	        Signals_109_5 AT %X45.5 : BOOL;
	        Signals_109_6 AT %X45.6 : BOOL;
	        Signals_109_7 AT %X45.7 : BOOL;
	        Signals_110_0 AT %X46.0 : BOOL;
	        Signals_110_1 AT %X46.1 : BOOL;
	        Signals_110_2 AT %X46.2 : BOOL;
	        Signals_110_3 AT %X46.3 : BOOL;
	        Signals_110_4 AT %X46.4 : BOOL;
	        Signals_110_5 AT %X46.5 : BOOL;
	        Signals_110_6 AT %X46.6 : BOOL;
	        Signals_110_7 AT %X46.7 : BOOL;
	        Signals_111_0 AT %X47.0 : BOOL;
	        Signals_111_1 AT %X47.1 : BOOL;
	        Signals_111_2 AT %X47.2 : BOOL;
	        Signals_111_3 AT %X47.3 : BOOL;
	        Signals_111_4 AT %X47.4 : BOOL;
	        Signals_111_5 AT %X47.5 : BOOL;
	        Signals_111_6 AT %X47.6 : BOOL;
	        Signals_111_7 AT %X47.7 : BOOL;
	        Signals_112_0 AT %X48.0 : BOOL;
	        Signals_112_1 AT %X48.1 : BOOL;
	        Signals_112_2 AT %X48.2 : BOOL;
	        Signals_112_3 AT %X48.3 : BOOL;
	        Signals_112_4 AT %X48.4 : BOOL;
	        Signals_112_5 AT %X48.5 : BOOL;
	        Signals_112_6 AT %X48.6 : BOOL;
	        Signals_112_7 AT %X48.7 : BOOL;
	        Signals_113_0 AT %X49.0 : BOOL;
	        Signals_113_1 AT %X49.1 : BOOL;
	        Signals_113_2 AT %X49.2 : BOOL;
	        Signals_113_3 AT %X49.3 : BOOL;
	        Signals_113_4 AT %X49.4 : BOOL;
	        Signals_113_5 AT %X49.5 : BOOL;
	        Signals_113_6 AT %X49.6 : BOOL;
	        Signals_113_7 AT %X49.7 : BOOL;
	        Signals_114_0 AT %X50.0 : BOOL;
	        Signals_114_1 AT %X50.1 : BOOL;
	        Signals_114_2 AT %X50.2 : BOOL;
	        Signals_114_3 AT %X50.3 : BOOL;
	        Signals_114_4 AT %X50.4 : BOOL;
	        Signals_114_5 AT %X50.5 : BOOL;
	        Signals_114_6 AT %X50.6 : BOOL;
	        Signals_114_7 AT %X50.7 : BOOL;
	        Signals_115_0 AT %X51.0 : BOOL;
	        Signals_115_1 AT %X51.1 : BOOL;
	        Signals_115_2 AT %X51.2 : BOOL;
	        Signals_115_3 AT %X51.3 : BOOL;
	        Signals_115_4 AT %X51.4 : BOOL;
	        Signals_115_5 AT %X51.5 : BOOL;
	        Signals_115_6 AT %X51.6 : BOOL;
	        Signals_115_7 AT %X51.7 : BOOL;
	        Signals_116_0 AT %X52.0 : BOOL;
	        Signals_116_1 AT %X52.1 : BOOL;
	        Signals_116_2 AT %X52.2 : BOOL;
	        Signals_116_3 AT %X52.3 : BOOL;
	        Signals_116_4 AT %X52.4 : BOOL;
	        Signals_116_5 AT %X52.5 : BOOL;
	        Signals_116_6 AT %X52.6 : BOOL;
	        Signals_116_7 AT %X52.7 : BOOL;
	        Signals_117_0 AT %X53.0 : BOOL;
	        Signals_117_1 AT %X53.1 : BOOL;
	        Signals_117_2 AT %X53.2 : BOOL;
	        Signals_117_3 AT %X53.3 : BOOL;
	        Signals_117_4 AT %X53.4 : BOOL;
	        Signals_117_5 AT %X53.5 : BOOL;
	        Signals_117_6 AT %X53.6 : BOOL;
	        Signals_117_7 AT %X53.7 : BOOL;
	        Signals_118_0 AT %X54.0 : BOOL;
	        Signals_118_1 AT %X54.1 : BOOL;
	        Signals_118_2 AT %X54.2 : BOOL;
	        Signals_118_3 AT %X54.3 : BOOL;
	        Signals_118_4 AT %X54.4 : BOOL;
	        Signals_118_5 AT %X54.5 : BOOL;
	        Signals_118_6 AT %X54.6 : BOOL;
	        Signals_118_7 AT %X54.7 : BOOL;
	        Signals_119_0 AT %X55.0 : BOOL;
	        Signals_119_1 AT %X55.1 : BOOL;
	        Signals_119_2 AT %X55.2 : BOOL;
	        Signals_119_3 AT %X55.3 : BOOL;
	        Signals_119_4 AT %X55.4 : BOOL;
	        Signals_119_5 AT %X55.5 : BOOL;
	        Signals_119_6 AT %X55.6 : BOOL;
	        Signals_119_7 AT %X55.7 : BOOL;
	        Signals_120_0 AT %X56.0 : BOOL;
	        Signals_120_1 AT %X56.1 : BOOL;
	        Signals_120_2 AT %X56.2 : BOOL;
	        Signals_120_3 AT %X56.3 : BOOL;
	        Signals_120_4 AT %X56.4 : BOOL;
	        Signals_120_5 AT %X56.5 : BOOL;
	        Signals_120_6 AT %X56.6 : BOOL;
	        Signals_120_7 AT %X56.7 : BOOL;
	        Signals_121_0 AT %X57.0 : BOOL;
	        Signals_121_1 AT %X57.1 : BOOL;
	        Signals_121_2 AT %X57.2 : BOOL;
	        Signals_121_3 AT %X57.3 : BOOL;
	        Signals_121_4 AT %X57.4 : BOOL;
	        Signals_121_5 AT %X57.5 : BOOL;
	        Signals_121_6 AT %X57.6 : BOOL;
	        Signals_121_7 AT %X57.7 : BOOL;
	        Signals_122_0 AT %X58.0 : BOOL;
	        Signals_122_1 AT %X58.1 : BOOL;
	        Signals_122_2 AT %X58.2 : BOOL;
	        Signals_122_3 AT %X58.3 : BOOL;
	        Signals_122_4 AT %X58.4 : BOOL;
	        Signals_122_5 AT %X58.5 : BOOL;
	        Signals_122_6 AT %X58.6 : BOOL;
	        Signals_122_7 AT %X58.7 : BOOL;
	        Signals_123_0 AT %X59.0 : BOOL;
	        Signals_123_1 AT %X59.1 : BOOL;
	        Signals_123_2 AT %X59.2 : BOOL;
	        Signals_123_3 AT %X59.3 : BOOL;
	        Signals_123_4 AT %X59.4 : BOOL;
	        Signals_123_5 AT %X59.5 : BOOL;
	        Signals_123_6 AT %X59.6 : BOOL;
	        Signals_123_7 AT %X59.7 : BOOL;
	        Signals_124_0 AT %X60.0 : BOOL;
	        Signals_124_1 AT %X60.1 : BOOL;
	        Signals_124_2 AT %X60.2 : BOOL;
	        Signals_124_3 AT %X60.3 : BOOL;
	        Signals_124_4 AT %X60.4 : BOOL;
	        Signals_124_5 AT %X60.5 : BOOL;
	        Signals_124_6 AT %X60.6 : BOOL;
	        Signals_124_7 AT %X60.7 : BOOL;
	        Signals_125_0 AT %X61.0 : BOOL;
	        Signals_125_1 AT %X61.1 : BOOL;
	        Signals_125_2 AT %X61.2 : BOOL;
	        Signals_125_3 AT %X61.3 : BOOL;
	        Signals_125_4 AT %X61.4 : BOOL;
	        Signals_125_5 AT %X61.5 : BOOL;
	        Signals_125_6 AT %X61.6 : BOOL;
	        Signals_125_7 AT %X61.7 : BOOL;
	        Signals_126_0 AT %X62.0 : BOOL;
	        Signals_126_1 AT %X62.1 : BOOL;
	        Signals_126_2 AT %X62.2 : BOOL;
	        Signals_126_3 AT %X62.3 : BOOL;
	        Signals_126_4 AT %X62.4 : BOOL;
	        Signals_126_5 AT %X62.5 : BOOL;
	        Signals_126_6 AT %X62.6 : BOOL;
	        Signals_126_7 AT %X62.7 : BOOL;
	        Signals_127_0 AT %X63.0 : BOOL;
	        Signals_127_1 AT %X63.1 : BOOL;
	        Signals_127_2 AT %X63.2 : BOOL;
	        Signals_127_3 AT %X63.3 : BOOL;
	        Signals_127_4 AT %X63.4 : BOOL;
	        Signals_127_5 AT %X63.5 : BOOL;
	        Signals_127_6 AT %X63.6 : BOOL;
	        Signals_127_7 AT %X63.7 : BOOL;
	    END_STRUCT;
	END_TYPE
